// Map values
SIR.Position := PositionName;
SIR.Code := Code;
SIR.TU_ID := TU_ID;
SIR.Counter1 := Counter1;
SIR.Counter2 := Counter2;
SIR.Counter3 := Counter3;
SIR.Counter4 := Counter4;
SIR.Counter5 := Counter5;
SIR.eReturnCode := eReturnCode;

// Forward to ITC
F_ITC_SendSIR := fbITC_Manager.M_SendData(
					meChannel	:= eChannelSrc,
					mMsgType	:= E_ITC_MsgTypeConv.SCANNER_INFORMATION_REPORT,
					mpData		:= ADR(SIR),
					mLen		:= SIZEOF(SIR));

END_FUNCTION

// ---- 20_Product/10_BCF/11_Conv/11_Com/11_ITC/F_ITC_SendSNR.TcPOU
FUNCTION F_ITC_SendSNR : BOOL
(**************************************************************************************
 * 	Application		:	BoxControl Framework
 *	Revision		:	$Revision: 404529 $
 *	Revision date	:	$Date: 2018-04-23 08:21:38 +0200 (Mo., 23 Apr 2018) $
 *	Last changed by	:	$Author: b7bolm $
 *	URL				:	$URL: http://almscdc.swisslog.com/repo/SWPD/Development/BoxControlFramework/20_Release/trunk/01_Software/BCF/BCF/JumpStart/20_Product/10_App/11_Com/10_Lib/10_Conv/11_ITC/F_ITC_SendSNR.TcPOU $
 *
 *	Purpose			:	Wrap message - SNR
 *
 * ------------------------------------------------------------------------------------
 *	Copyright Swisslog [IP AG], Switzerland. All rights reserved.
 * 
 * ------------------------------------------------------------------------------------
 *	
 * 	Revision History: 
 *
 * 	VERSION			DATE			INITIALS			DESCRIPTION
 *	0.1				01.01.2001		swl					Example
 *
 **************************************************************************************)
VAR_INPUT
	eChannelSrc		: E_MFCS_Channel; // Source communicaton channel	
	PositionName	: STRING(Conveyor.POSITION_STRINGLENGTH); // Position
	TU_ID			: STRING(Conveyor.TU_ID_STRINGLENGTH); // TU ID
	eInfoCode		: E_ErrorConv; // Info Code
END_VAR
VAR
	SNR				: ST_ITC_SNR; 
END_VAR

// Map values
SNR.Position := PositionName;
SNR.TU_ID := TU_ID;
SNR.InfoCode := eInfoCode;

// Forward to ITC
F_ITC_SendSNR := fbITC_Manager.M_SendData(
					meChannel	:= eChannelSrc,
					mMsgType	:= E_ITC_MsgTypeConv.SCANNER_NO_READ_REPORT,
					mpData		:= ADR(SNR),
					mLen		:= SIZEOF(SNR));

END_FUNCTION

// ---- 20_Product/10_BCF/11_Conv/11_Com/11_ITC/F_ITC_SendTDR.TcPOU
FUNCTION F_ITC_SendTDR : BOOL
(**************************************************************************************
 * 	Application		:	BoxControl Framework
 *	Revision		:	$Revision: 404529 $
 *	Revision date	:	$Date: 2018-04-23 08:21:38 +0200 (Mo., 23 Apr 2018) $
 *	Last changed by	:	$Author: b7bolm $
 *	URL				:	$URL: http://almscdc.swisslog.com/repo/SWPD/Development/BoxControlFramework/20_Release/trunk/01_Software/BCF/BCF/JumpStart/20_Product/10_App/11_Com/10_Lib/10_Conv/11_ITC/F_ITC_SendTDR.TcPOU $
 *
 *	Purpose			:	Wrap message - TDR
 *
 * ------------------------------------------------------------------------------------
 *	Copyright Swisslog [IP AG], Switzerland. All rights reserved.
 * 
 * ------------------------------------------------------------------------------------
 *	
 * 	Revision History: 
 *
 * 	VERSION			DATE			INITIALS			DESCRIPTION
 *	0.1				01.01.2001		swl					Example
 *
 **************************************************************************************)
VAR_INPUT
	eChannelSrc		: E_MFCS_Channel; // Source communicaton channel	
	PositionName	: STRING(Conveyor.POSITION_STRINGLENGTH); // SIS MM-GGG-EEEE-FF-Z
	TU_ID			: STRING(Conveyor.TU_ID_STRINGLENGTH); // 18 Digit SSID
	AssignmentID	: UDINT; // assignment id
	MsgSequence		: INT; // MSG Sequence
	eReturnCode		: E_ErrorConv; // Return code
END_VAR
VAR
	TDR				: ST_ITC_TDR; 
END_VAR

// Map values
TDR.Position := PositionName;
TDR.TU_ID := TU_ID;
TDR.AssignmentID := AssignmentID;
TDR.MsgSequence := MsgSequence;
TDR.ReturnCode := eReturnCode;

// Forward to ITC
F_ITC_SendTDR := fbITC_Manager.M_SendData(
					meChannel	:= eChannelSrc,
					mMsgType	:= E_ITC_MsgTypeConv.TASK_DELETE_REPORT,
					mpData		:= ADR(TDR),
					mLen		:= SIZEOF(TDR));

END_FUNCTION

// ---- 20_Product/10_BCF/11_Conv/11_Com/11_ITC/F_ITC_SendTTC.TcPOU
FUNCTION F_ITC_SendTTC : BOOL
(**************************************************************************************
 * 	Application		:	BoxControl Framework
 *	Revision		:	$Revision: 404529 $
 *	Revision date	:	$Date: 2018-04-23 08:21:38 +0200 (Mo., 23 Apr 2018) $
 *	Last changed by	:	$Author: b7bolm $
 *	URL				:	$URL: http://almscdc.swisslog.com/repo/SWPD/Development/BoxControlFramework/20_Release/trunk/01_Software/BCF/BCF/JumpStart/20_Product/10_App/11_Com/10_Lib/10_Conv/11_ITC/F_ITC_SendTTC.TcPOU $
 *
 *	Purpose			:	Wrap message - TTC
 *
 * ------------------------------------------------------------------------------------
 *	Copyright Swisslog [IP AG], Switzerland. All rights reserved.
 * 
 * ------------------------------------------------------------------------------------
 *	
 * 	Revision History: 
 *
 * 	VERSION			DATE			INITIALS			DESCRIPTION
 *	0.1				01.01.2001		swl					Example
 *
 **************************************************************************************)
VAR_INPUT
	eChannelSrc		: E_MFCS_Channel; // Source communicaton channel		
	PositionName	: STRING(Conveyor.POSITION_STRINGLENGTH); // Position
	TU_DataIndex	: DINT; // TU-DataIndex
	MsgSequence		: INT; // Assignment message sequence
	TU_ID			: STRING(Conveyor.TU_ID_STRINGLENGTH); // 18 Digit SSID
	AssignmentID	: UDINT; // assignment id
	eReturnCode		: E_ErrorConv; // Return code
END_VAR
VAR
	TTC				: ST_ITC_TTC; 
END_VAR

// Map values
TTC.Position := PositionName;
TTC.TU_DataIndex := TU_DataIndex;
TTC.MsgSequence := MsgSequence;
TTC.TU_ID := TU_ID;
TTC.AssignmentID := AssignmentID;
TTC.ReturnCode := eReturnCode;

// Forward to ITC
F_ITC_SendTTC := fbITC_Manager.M_SendData(
					meChannel	:= eChannelSrc,
					mMsgType	:= E_ITC_MsgTypeConv.TRANSPORT_TASK_COMPLETE,
					mpData		:= ADR(TTC),
					mLen		:= SIZEOF(TTC));

END_FUNCTION

// ---- 20_Product/10_BCF/11_Conv/11_Com/11_ITC/F_ITC_SendTTQ.TcPOU
FUNCTION F_ITC_SendTTQ : BOOL
(**************************************************************************************
 * 	Application		:	BoxControl Framework
 *	Revision		:	$Revision: 404529 $
 *	Revision date	:	$Date: 2018-04-23 08:21:38 +0200 (Mo., 23 Apr 2018) $
 *	Last changed by	:	$Author: b7bolm $
 *	URL				:	$URL: http://almscdc.swisslog.com/repo/SWPD/Development/BoxControlFramework/20_Release/trunk/01_Software/BCF/BCF/JumpStart/20_Product/10_App/11_Com/10_Lib/10_Conv/11_ITC/F_ITC_SendTTQ.TcPOU $
 *
 *	Purpose			:	Wrap message - TTQ
 *
 * ------------------------------------------------------------------------------------
 *	Copyright Swisslog [IP AG], Switzerland. All rights reserved.
 * 
 * ------------------------------------------------------------------------------------
 *	
 * 	Revision History: 
 *
 * 	VERSION			DATE			INITIALS			DESCRIPTION
 *	0.1				01.01.2001		swl					Example
 *
 **************************************************************************************)
VAR_INPUT
	eChannelSrc		: E_MFCS_Channel; // Source communicaton channel	
	PositionName	: STRING(Conveyor.POSITION_STRINGLENGTH); // Position
	TU_DataIndex	: DINT; // TU-DataIndex
	TU_ID			: STRING(Conveyor.TU_ID_STRINGLENGTH); // TU ID
	NbrOfTT			: INT; // Number of TT's
	Label			: STRING(Conveyor.LABEL_LENGTH); // Label length
END_VAR
VAR
	TTQ				: ST_ITC_TTQ; 
END_VAR

// Map values
TTQ.Position := PositionName;
TTQ.TU_DataIndex := TU_DataIndex;
TTQ.TU_ID := TU_ID;
TTQ.NbrOfTT := NbrOfTT;
TTQ.Label := Label;

// Forward to ITC
F_ITC_SendTTQ := fbITC_Manager.M_SendData(
					meChannel	:= eChannelSrc,
					mMsgType	:= E_ITC_MsgTypeConv.TRANSPORT_TASK_REQUEST,
					mpData		:= ADR(TTQ),
					mLen		:= SIZEOF(TTQ));

END_FUNCTION

// ---- 20_Product/10_BCF/11_Conv/11_Com/11_ITC/F_ITC_SendTUR.TcPOU
FUNCTION F_ITC_SendTUR : BOOL
(**************************************************************************************
 * 	Application		:	BoxControl Framework
 *	Revision		:	$Revision: 416339 $
 *	Revision date	:	$Date: 2018-10-31 13:50:31 +0100 (Wed, 31 Oct 2018) $
 *	Last changed by	:	$Author: b7bolm $
 *	URL				:	$URL: http://almscdc.swisslog.com/repo/SWPD/Development/BoxControlFramework/20_Release/branches/R1.5.x/01_Software/BCF/BCF/JumpStart/20_Product/10_App/11_Com/10_Lib/10_Conv/11_ITC/F_ITC_SendTUR.TcPOU $
 *
 *	Purpose			:	Wrap message - TUR
 *
 * ------------------------------------------------------------------------------------
 *	Copyright Swisslog [IP AG], Switzerland. All rights reserved.
 * 
 * ------------------------------------------------------------------------------------
 *	
 * 	Revision History: 
 *
 * 	VERSION			DATE			INITIALS			DESCRIPTION
 *	0.1				01.01.2001		swl					Example
 *
 **************************************************************************************)
VAR_INPUT
	eChannelSrc				: E_MFCS_Channel; // Source communicaton channel	
	LastPositionName		: STRING(Conveyor.POSITION_STRINGLENGTH); // Position
	TU_DataIndex			: DINT; // Data index
	TU_ID					: STRING(Conveyor.TU_ID_STRINGLENGTH); // TU ID
	TU_Type					: INT; // TU Type
	AssignmentID			: UDINT; // Assignment ID
	Length					: INT; // Length
	Width					: INT; // Width
	Height					: INT; // Height
	Weight					: DINT; // Weight
	Orientation				: STRING(Conveyor.ORIENTATION_STRINGLENGTH); // 3 Digit orientation
	TU_Parameter			: INT; // TU Parameter
	IO_Data					: INT; // IO Data
	LowerLimit				: DINT; // Lower Limit
	UpperLimit				: DINT; // Upper Limit
	Sequence				: ULINT; // Global sequence identifier
	SubSequence				: DINT; // Position in the sequence
	SequenceSize			: DINT; // Number of TU's in the sequence
	GroupID					: ULINT; // Global group identifier 
	GroupSize				: DINT; // Number of TU's in the group ID
	DestinationSlot         : INT; // Logical sub destination of destination
	eReturnCode				: E_ErrorConv; // Return code
	NumberOfDestinations	: INT; // Number of Destinations
	Destination				: ARRAY [1..Conveyor.NUMBER_OF_DESTINATIONS] OF STRING(Conveyor.POSITION_STRINGLENGTH); // Array of SIS Destinations
END_VAR
VAR
	TUR						: ST_ITC_TUR; 
END_VAR

// Map values
TUR.Position := LastPositionName;
TUR.TU_DataIndex := TU_DataIndex;
TUR.TU_ID := TU_ID;
TUR.TU_Type := TU_Type;
TUR.AssignmentID := AssignmentID;
TUR.Length := Length;
TUR.Width := Width;
TUR.Height := Height;
TUR.Weight := Weight;
TUR.Orientation := Orientation;
TUR.TU_Parameter := TU_Parameter;
TUR.IO_Data := IO_Data;
TUR.LowerLimit := LowerLimit;
TUR.UpperLimit := UpperLimit;
TUR.Sequence := Sequence;
TUR.SubSequence := SubSequence;
TUR.SequenceSize := SequenceSize;
TUR.GroupID := GroupID;
TUR.GroupSize := GroupSize;
TUR.DestinationSlot := DestinationSlot;
TUR.ReturnCode := eReturnCode;
TUR.NumberOfDestinations := NumberOfDestinations;
TUR.Destination := Destination;

// Forward to ITC
F_ITC_SendTUR := fbITC_Manager.M_SendData(
					meChannel	:= eChannelSrc,
					mMsgType	:= E_ITC_MsgTypeConv.TRANSPORT_UNIT_REPORT,
					mpData		:= ADR(TUR),
					mLen		:= SIZEOF(TUR));

END_FUNCTION

// ---- 20_Product/10_BCF/11_Conv/11_Com/13_Sub-Sub/FB_STI_SendReceiveTU_Data_6_0.TcPOU
FUNCTION_BLOCK FB_STI_SendReceiveTU_Data_6_0
(**************************************************************************************
 * 	Application		:	BoxControl Framework
 *	Revision		:	$Revision: 404529 $
 *	Revision date	:	$Date: 2018-04-23 08:21:38 +0200 (Mo., 23 Apr 2018) $
 *	Last changed by	:	$Author: b7bolm $
 *	URL				:	$URL: http://almscdc.swisslog.com/repo/SWPD/Development/BoxControlFramework/20_Release/trunk/01_Software/BCF/BCF/JumpStart/20_Product/10_App/11_Com/10_Lib/10_Conv/13_Sub-Sub/FB_STI_SendReceiveTU_Data_6_0.TcPOU $
 *
 *	Purpose			:	Sends and Receive TU-data to/from other SubSystem via TTA
 *
 * ------------------------------------------------------------------------------------
 *	Copyright Swisslog [IP AG], Switzerland. All rights reserved.
 * 
 * ------------------------------------------------------------------------------------
 *	
 * 	Revision History: 
 *
 * 	VERSION			DATE			INITIALS			DESCRIPTION
 *	0.1				01.01.2001		swl					Example
 *
 **************************************************************************************)
VAR_INPUT
	PositionSubSystem		: STRING(SIS_6_0.POSITION_STRINGLENGTH); // SIS-Position of SubSystem
	ConfigSIS_MsgManager	: ST_CFG_SIS_MsgManager_6_0; // Configuration
END_VAR
VAR
	Init					: BOOL := FALSE; // Instance is initialized
	fbMFCS_SIS_Sub			: FB_SIS_MsgManager_6_0; // Instance of SIS-driver
	TTA						: ST_TTA_6_0; // TTA structure
	SendTelegram			: ARRAY [1..MAX_STREAM_LENGTH] OF BYTE; // Send telegram
END_VAR
VAR CONSTANT
	MAX_STREAM_LENGTH		: UDINT := 30000; // Number of bytes of one message
END_VAR

(**************************************************************************************************************
   Initialization
***************************************************************************************************************)
A_Init();


(**************************************************************************************************************
   Call SIS-driver
***************************************************************************************************************)
fbMFCS_SIS_Sub.M_CallCommunicationService();

ACTION A_Init:
(**************************************************************************************
 * 	NAME		A_Init
 * 	FUNCTION	Initialize FB
 **************************************************************************************)
// If instance is not initialized or init is forced
IF NOT Init THEN
	
	// Activate configuration
	fbMFCS_SIS_Sub.Config := ConfigSIS_MsgManager;
	
	// Init done
    Init := TRUE;
END_IF
END_ACTION

METHOD M_SendTTA : BOOL
(**************************************************************************************
 * 	Application		:	BoxControl Framework
 *	Revision		:	$Revision: 404529 $
 *	Revision date	:	$Date: 2018-04-23 08:21:38 +0200 (Mo., 23 Apr 2018) $
 *	Last changed by	:	$Author: b7bolm $
 *	URL				:	$URL: http://almscdc.swisslog.com/repo/SWPD/Development/BoxControlFramework/20_Release/trunk/01_Software/BCF/BCF/JumpStart/20_Product/10_App/11_Com/10_Lib/10_Conv/13_Sub-Sub/FB_STI_SendReceiveTU_Data_6_0.TcPOU $
 *
 *	Purpose			:	Send TTA
 *
 * ------------------------------------------------------------------------------------
 *	Copyright Swisslog [IP AG], Switzerland. All rights reserved.
 * 
 * ------------------------------------------------------------------------------------
 *	
 * 	Revision History: 
 *
 * 	VERSION			DATE			INITIALS			DESCRIPTION
 *	0.1				01.01.2001		swl					Example
 *
 **************************************************************************************)
VAR_INPUT
 	mTU_DataIndex		: DINT;
END_VAR
VAR
	mIdx				: INT;
	mWritePointer		: UDINT;
END_VAR
(**************************************************************************************************************
 	Formatting data
***************************************************************************************************************)
TTA.Position := F_StuffString(
					InputString 	:= PositionSubSystem, 
					StringLength	:= SIS_6_0.POSITION_STRINGLENGTH, 
					StuffCharacter 	:= '0',
					LeftAligned		:= FALSE);
					
TTA.TU_DataIndex := F_StuffString(
					InputString 	:= '0', 
					StringLength	:= SIS_6_0.TU_DATAINDEX_STRINGLENGTH, 
					StuffCharacter 	:= '0',
					LeftAligned		:= FALSE);
					
TTA.MsgSequence := F_StuffString(
					InputString 	:= '0', 
					StringLength	:= SIS_6_0.MSG_SEQUENCE_STRINGLENGTH, 
					StuffCharacter 	:= '0',
					LeftAligned		:= FALSE);

TTA.TU_ID := F_StuffString(
					InputString 	:= TU_DataTable[mTU_DataIndex].TU_ID.ASCII, 
					StringLength	:= SIS_6_0.TU_ID_STRINGLENGTH, 
					StuffCharacter 	:= ' ',
					LeftAligned		:= FALSE);
					
TTA.TU_Type := F_StuffString(
					InputString 	:= INT_TO_STRING(TU_DataTable[mTU_DataIndex].DataSet.TU_Type), 
					StringLength	:= SIS_6_0.TU_TYPE_STRINGLENGTH, 
					StuffCharacter 	:= '0',
					LeftAligned		:= FALSE);
					
TTA.AssignmentID := F_StuffString(
					InputString 	:= UDINT_TO_STRING(TU_DataTable[mTU_DataIndex].AssignmentID), 
					StringLength	:= SIS_6_0.ASSIGNMENT_ID_STRINGLENGTH, 
					StuffCharacter 	:= '0',
					LeftAligned		:= FALSE);
					
TTA.Length := F_StuffString(
					InputString 	:= INT_TO_STRING(TU_DataTable[mTU_DataIndex].DataSet.Dimension.Length), 
					StringLength	:= SIS_6_0.DIMENSIONS, 
					StuffCharacter 	:= '0',
					LeftAligned		:= FALSE);
					
TTA.Width := F_StuffString(
					InputString 	:= INT_TO_STRING(TU_DataTable[mTU_DataIndex].DataSet.Dimension.Width), 
					StringLength	:= SIS_6_0.DIMENSIONS, 
					StuffCharacter 	:= '0',
					LeftAligned		:= FALSE);
					
TTA.Height := F_StuffString(
					InputString 	:= INT_TO_STRING(TU_DataTable[mTU_DataIndex].DataSet.Dimension.Height), 
					StringLength	:= SIS_6_0.DIMENSIONS, 
					StuffCharacter 	:= '0',
					LeftAligned		:= FALSE);
					
TTA.Weight := F_StuffString(
					InputString 	:= DINT_TO_STRING(TU_DataTable[mTU_DataIndex].DataSet.Dimension.Weight), 
					StringLength	:= SIS_6_0.TTA_WEIGHT, 
					StuffCharacter 	:= '0',
					LeftAligned		:= FALSE);
					
TTA.Orientation := F_StuffString(
					InputString 	:= TU_DataTable[mTU_DataIndex].DataSet.Orientation, 
					StringLength	:= SIS_6_0.TTA_ORIENTATION, 
					StuffCharacter 	:= '0',
					LeftAligned		:= FALSE);

TTA.TU_Parameter := F_StuffString(
					InputString 	:= INT_TO_STRING(TU_DataTable[mTU_DataIndex].DataSet.TU_Parameter), 
					StringLength	:= SIS_6_0.TTA_TU_PARAMETER, 
					StuffCharacter 	:= '0',
					LeftAligned		:= FALSE);
					
TTA.IO_Data := F_StuffString(
					InputString 	:= INT_TO_STRING(TU_DataTable[mTU_DataIndex].DataSet.IO_Data), 
					StringLength	:= SIS_6_0.TTA_IO_DATA_STRINGLENGTH, 
					StuffCharacter 	:= '0',
					LeftAligned		:= FALSE);
					
TTA.LowerLimit := F_StuffString(
					InputString 	:= DINT_TO_STRING(TU_DataTable[mTU_DataIndex].DataSet.LowerLimit), 
					StringLength	:= SIS_6_0.TTA_LOWER_LIMIT_STRINGLENGTH, 
					StuffCharacter 	:= '0',
					LeftAligned		:= FALSE);
					
TTA.UpperLimit := F_StuffString(
					InputString 	:= DINT_TO_STRING(TU_DataTable[mTU_DataIndex].DataSet.UpperLimit), 
					StringLength	:= SIS_6_0.TTA_UPPER_LIMIT_STRINGLENGTH, 
					StuffCharacter 	:= '0',
					LeftAligned		:= FALSE);
					
TTA.GroupInfo := F_StuffString(
					InputString 	:= ULINT_TO_STRING(TU_DataTable[mTU_DataIndex].DataSet.GroupID), 
					StringLength	:= SIS_6_0.TTA_GROUPINFO_STRINGLENGTH, 
					StuffCharacter 	:= '0',
					LeftAligned		:= FALSE);
					
TTA.Sequence := F_StuffString(
					InputString 	:= ULINT_TO_STRING(TU_DataTable[mTU_DataIndex].DataSet.Sequence), 
					StringLength	:= SIS_6_0.TTA_SEQUENCE_STRINGLENGTH, 
					StuffCharacter 	:= '0',
					LeftAligned		:= FALSE);
					
TTA.NumberInSequence := F_StuffString(
					InputString 	:= DINT_TO_STRING(TU_DataTable[mTU_DataIndex].DataSet.SubSequence), 
					StringLength	:= SIS_6_0.TTA_NO_IN_SEQUENCE_STRINGLENGTH, 
					StuffCharacter 	:= '0',
					LeftAligned		:= FALSE);
					
TTA.NumberOfDestinations := F_StuffString(
					InputString 	:= INT_TO_STRING(TU_DataTable[mTU_DataIndex].DataSet.NumberOfDest), 
					StringLength	:= SIS_6_0.TTA_NO_OF_DESTINATIONS_STRINGLENGTH, 
					StuffCharacter 	:= '0',
					LeftAligned		:= FALSE);
					
FOR mIdx := 1 TO TU_DataTable[mTU_DataIndex].DataSet.NumberOfDest DO
	TTA.Destination[mIdx] := F_StuffString(
					InputString 	:= TU_DataTable[mTU_DataIndex].Destination[mIdx].PositionName, 
					StringLength	:= SIS_6_0.POSITION_STRINGLENGTH, 
					StuffCharacter 	:= '0',
					LeftAligned		:= FALSE);
END_FOR
					
					
(**************************************************************************************************************
 	Build string and add to Base Driver
***************************************************************************************************************)
MEMSET(destAddr := ADR(SendTelegram), 0, SIZEOF(SendTelegram));
mWritePointer := 0;

F_AssembleByteStream(
	pSrc 			:= ADR('TTA'), 
	SrcLen 			:= 3, 
	pDest 			:= ADR(SendTelegram), 
	DestLen 		:= SIZEOF(SendTelegram), 
	WritePointer	:= mWritePointer);
	
F_AssembleByteStream(
	pSrc 			:= ADR(TTA.Position), 
	SrcLen 			:= INT_TO_UDINT(LEN(TTA.Position)), 
	pDest 			:= ADR(SendTelegram), 
	DestLen 		:= SIZEOF(SendTelegram), 
	WritePointer	:= mWritePointer);
	
F_AssembleByteStream(
	pSrc 			:= ADR(TTA.TU_DataIndex), 
	SrcLen 			:= INT_TO_UDINT(LEN(TTA.TU_DataIndex)), 
	pDest 			:= ADR(SendTelegram), 
	DestLen 		:= SIZEOF(SendTelegram), 
	WritePointer	:= mWritePointer);
	
F_AssembleByteStream(
	pSrc 			:= ADR(TTA.MsgSequence), 
	SrcLen 			:= INT_TO_UDINT(LEN(TTA.MsgSequence)), 
	pDest 			:= ADR(SendTelegram), 
	DestLen 		:= SIZEOF(SendTelegram), 
	WritePointer	:= mWritePointer);
	
F_AssembleByteStream(
	pSrc 			:= ADR(TTA.TU_ID), 
	SrcLen 			:= INT_TO_UDINT(LEN(TTA.TU_ID)), 
	pDest 			:= ADR(SendTelegram), 
	DestLen 		:= SIZEOF(SendTelegram), 
	WritePointer	:= mWritePointer);
	
F_AssembleByteStream(
	pSrc 			:= ADR(TTA.TU_Type), 
	SrcLen 			:= INT_TO_UDINT(LEN(TTA.TU_Type)), 
	pDest 			:= ADR(SendTelegram), 
	DestLen 		:= SIZEOF(SendTelegram), 
	WritePointer	:= mWritePointer);	
	
F_AssembleByteStream(
	pSrc 			:= ADR(TTA.AssignmentID), 
	SrcLen 			:= INT_TO_UDINT(LEN(TTA.AssignmentID)), 
	pDest 			:= ADR(SendTelegram), 
	DestLen 		:= SIZEOF(SendTelegram), 
	WritePointer	:= mWritePointer);		
	
F_AssembleByteStream(
	pSrc 			:= ADR(TTA.Length), 
	SrcLen 			:= INT_TO_UDINT(LEN(TTA.Length)), 
	pDest 			:= ADR(SendTelegram), 
	DestLen 		:= SIZEOF(SendTelegram), 
	WritePointer	:= mWritePointer);

F_AssembleByteStream(
	pSrc 			:= ADR(TTA.Width), 
	SrcLen 			:= INT_TO_UDINT(LEN(TTA.Width)), 
	pDest 			:= ADR(SendTelegram), 
	DestLen 		:= SIZEOF(SendTelegram), 
	WritePointer	:= mWritePointer);
	
F_AssembleByteStream(
	pSrc 			:= ADR(TTA.Height), 
	SrcLen 			:= INT_TO_UDINT(LEN(TTA.Height)), 
	pDest 			:= ADR(SendTelegram), 
	DestLen 		:= SIZEOF(SendTelegram), 
	WritePointer	:= mWritePointer);
	
F_AssembleByteStream(
	pSrc 			:= ADR(TTA.Weight), 
	SrcLen 			:= INT_TO_UDINT(LEN(TTA.Weight)), 
	pDest 			:= ADR(SendTelegram), 
	DestLen 		:= SIZEOF(SendTelegram), 
	WritePointer	:= mWritePointer);
		
F_AssembleByteStream(
	pSrc 			:= ADR(TTA.Orientation), 
	SrcLen 			:= INT_TO_UDINT(LEN(TTA.Orientation)), 
	pDest 			:= ADR(SendTelegram), 
	DestLen 		:= SIZEOF(SendTelegram), 
	WritePointer	:= mWritePointer);
	
F_AssembleByteStream(
	pSrc 			:= ADR(TTA.TU_Parameter), 
	SrcLen 			:= INT_TO_UDINT(LEN(TTA.TU_Parameter)), 
	pDest 			:= ADR(SendTelegram), 
	DestLen 		:= SIZEOF(SendTelegram), 
	WritePointer	:= mWritePointer);	
	
F_AssembleByteStream(
	pSrc 			:= ADR(TTA.IO_Data), 
	SrcLen 			:= INT_TO_UDINT(LEN(TTA.IO_Data)), 
	pDest 			:= ADR(SendTelegram), 
	DestLen 		:= SIZEOF(SendTelegram), 
	WritePointer	:= mWritePointer);
	
F_AssembleByteStream(
	pSrc 			:= ADR(TTA.LowerLimit), 
	SrcLen 			:= INT_TO_UDINT(LEN(TTA.LowerLimit)), 
	pDest 			:= ADR(SendTelegram), 
	DestLen 		:= SIZEOF(SendTelegram), 
	WritePointer	:= mWritePointer);
	
F_AssembleByteStream(
	pSrc 			:= ADR(TTA.UpperLimit), 
	SrcLen 			:= INT_TO_UDINT(LEN(TTA.UpperLimit)), 
	pDest 			:= ADR(SendTelegram), 
	DestLen 		:= SIZEOF(SendTelegram), 
	WritePointer	:= mWritePointer);
	
F_AssembleByteStream(
	pSrc 			:= ADR(TTA.GroupInfo), 
	SrcLen 			:= INT_TO_UDINT(LEN(TTA.GroupInfo)), 
	pDest 			:= ADR(SendTelegram), 
	DestLen 		:= SIZEOF(SendTelegram), 
	WritePointer	:= mWritePointer);
	
F_AssembleByteStream(
	pSrc 			:= ADR(TTA.Sequence), 
	SrcLen 			:= INT_TO_UDINT(LEN(TTA.Sequence)), 
	pDest 			:= ADR(SendTelegram), 
	DestLen 		:= SIZEOF(SendTelegram), 
	WritePointer	:= mWritePointer);
	
F_AssembleByteStream(
	pSrc 			:= ADR(TTA.NumberInSequence), 
	SrcLen 			:= INT_TO_UDINT(LEN(TTA.NumberInSequence)), 
	pDest 			:= ADR(SendTelegram), 
	DestLen 		:= SIZEOF(SendTelegram), 
	WritePointer	:= mWritePointer);	

F_AssembleByteStream(
	pSrc 			:= ADR(TTA.NumberOfDestinations), 
	SrcLen 			:= INT_TO_UDINT(LEN(TTA.NumberOfDestinations)), 
	pDest 			:= ADR(SendTelegram), 
	DestLen 		:= SIZEOF(SendTelegram), 
	WritePointer	:= mWritePointer);	

FOR mIdx := 1 TO TU_DataTable[mTU_DataIndex].DataSet.NumberOfDest DO
	F_AssembleByteStream(
		pSrc 			:= ADR(TTA.Destination[mIdx]), 
		SrcLen 			:= INT_TO_UDINT(LEN(TTA.Destination[mIdx])), 
		pDest 			:= ADR(SendTelegram), 
		DestLen 		:= SIZEOF(SendTelegram), 
		WritePointer	:= mWritePointer);	
END_FOR	

M_SendTTA := fbMFCS_SIS_Sub.M_SendAppData(pData := ADR(SendTelegram), DataLen := mWritePointer);
END_METHOD

END_FUNCTION_BLOCK

// ---- 20_Product/10_BCF/11_Conv/11_Com/13_Sub-Sub/FB_STI_SendReceiveTU_Data_6_1.TcPOU
FUNCTION_BLOCK FB_STI_SendReceiveTU_Data_6_1
(**************************************************************************************
 * 	Application		:	BoxControl Framework
 *	Revision		:	$Revision: 404529 $
 *	Revision date	:	$Date: 2018-04-23 08:21:38 +0200 (Mo., 23 Apr 2018) $
 *	Last changed by	:	$Author: b7bolm $
 *	URL				:	$URL: http://almscdc.swisslog.com/repo/SWPD/Development/BoxControlFramework/20_Release/trunk/01_Software/BCF/BCF/JumpStart/20_Product/10_App/11_Com/10_Lib/10_Conv/13_Sub-Sub/FB_STI_SendReceiveTU_Data_6_1.TcPOU $
 *
 *	Purpose			:	Sends and Receive TU-data to/from other SubSystem via TTA
 *
 * ------------------------------------------------------------------------------------
 *	Copyright Swisslog [IP AG], Switzerland. All rights reserved.
 * 
 * ------------------------------------------------------------------------------------
 *	
 * 	Revision History: 
 *
 * 	VERSION			DATE			INITIALS			DESCRIPTION
 *	0.1				01.01.2001		swl					Example
 *
 **************************************************************************************)
VAR_INPUT
	PositionSubSystem		: STRING(SIS_6_1.POSITION_STRINGLENGTH); // SIS-Position of SubSystem
	ConfigSIS_MsgManager	: ST_CFG_SIS_MsgManager_6_1; // Configuration
END_VAR
VAR
	Init					: BOOL := FALSE; // Instance is initialized
	fbMFCS_SIS_Sub			: FB_SIS_MsgManager_6_1; // Instance of SIS-driver
	TTA						: ST_TTA_6_1; // TTA structure
	SendTelegram			: ARRAY [1..MAX_STREAM_LENGTH] OF BYTE; // Send telegram
END_VAR
VAR CONSTANT
	MAX_STREAM_LENGTH		: UDINT := 30000; // Number of bytes of one message
END_VAR

(**************************************************************************************************************
   Initialization
***************************************************************************************************************)
A_Init();


(**************************************************************************************************************
   Call SIS-driver
***************************************************************************************************************)
fbMFCS_SIS_Sub.M_CallCommunicationService();

ACTION A_Init:
(**************************************************************************************
 * 	NAME		A_Init
 * 	FUNCTION	Initialize FB
 **************************************************************************************)
// If instance is not initialized or init is forced
IF NOT Init THEN
	
	// Activate configuration
	fbMFCS_SIS_Sub.Config := ConfigSIS_MsgManager;
	
	// Init done
    Init := TRUE;
END_IF
END_ACTION

METHOD M_SendTTA : BOOL
(**************************************************************************************
 * 	Application		:	BoxControl Framework
 *	Revision		:	$Revision: 404529 $
 *	Revision date	:	$Date: 2018-04-23 08:21:38 +0200 (Mo., 23 Apr 2018) $
 *	Last changed by	:	$Author: b7bolm $
 *	URL				:	$URL: http://almscdc.swisslog.com/repo/SWPD/Development/BoxControlFramework/20_Release/trunk/01_Software/BCF/BCF/JumpStart/20_Product/10_App/11_Com/10_Lib/10_Conv/13_Sub-Sub/FB_STI_SendReceiveTU_Data_6_1.TcPOU $
 *
 *	Purpose			:	Send TTA
 *
 * ------------------------------------------------------------------------------------
 *	Copyright Swisslog [IP AG], Switzerland. All rights reserved.
 * 
 * ------------------------------------------------------------------------------------
 *	
 * 	Revision History: 
 *
 * 	VERSION			DATE			INITIALS			DESCRIPTION
 *	0.1				01.01.2001		swl					Example
 *
 **************************************************************************************)
VAR_INPUT
 	mTU_DataIndex		: DINT;
END_VAR
VAR
	mIdx				: INT;
	mWritePointer		: UDINT;
END_VAR
(**************************************************************************************************************
 	Formatting data
***************************************************************************************************************)
TTA.Position := F_StuffString(
					InputString 	:= PositionSubSystem, 
					StringLength	:= SIS_6_1.POSITION_STRINGLENGTH, 
					StuffCharacter 	:= '0',
					LeftAligned		:= FALSE);
					
TTA.TU_DataIndex := F_StuffString(
						InputString 	:= '0', 
						StringLength	:= SIS_6_1.TU_DATAINDEX_STRINGLENGTH, 
						StuffCharacter 	:= '0',
						LeftAligned		:= FALSE);
					
TTA.MsgSequence := F_StuffString(
					InputString 	:= '0', 
					StringLength	:= SIS_6_1.MSG_SEQUENCE_STRINGLENGTH, 
					StuffCharacter 	:= '0',
					LeftAligned		:= FALSE);

TTA.TU_ID := F_StuffString(
				InputString 	:= TU_DataTable[mTU_DataIndex].TU_ID.ASCII, 
				StringLength	:= SIS_6_1.TU_ID_STRINGLENGTH, 
				StuffCharacter 	:= ' ',
				LeftAligned		:= FALSE);
					
TTA.TU_Type := F_StuffString(
				InputString 	:= INT_TO_STRING(TU_DataTable[mTU_DataIndex].DataSet.TU_Type), 
				StringLength	:= SIS_6_1.TU_TYPE_STRINGLENGTH, 
				StuffCharacter 	:= '0',
				LeftAligned		:= FALSE);
					
TTA.AssignmentID := F_StuffString(
						InputString 	:= UDINT_TO_STRING(TU_DataTable[mTU_DataIndex].AssignmentID), 
						StringLength	:= SIS_6_1.ASSIGNMENT_ID_STRINGLENGTH, 
						StuffCharacter 	:= '0',
						LeftAligned		:= FALSE);
					
TTA.Length := F_StuffString(
				InputString 	:= INT_TO_STRING(TU_DataTable[mTU_DataIndex].DataSet.Dimension.Length), 
				StringLength	:= SIS_6_1.DIMENSIONS, 
				StuffCharacter 	:= '0',
				LeftAligned		:= FALSE);
					
TTA.Width := F_StuffString(
				InputString 	:= INT_TO_STRING(TU_DataTable[mTU_DataIndex].DataSet.Dimension.Width), 
				StringLength	:= SIS_6_1.DIMENSIONS, 
				StuffCharacter 	:= '0',
				LeftAligned		:= FALSE);
					
TTA.Height := F_StuffString(
				InputString 	:= INT_TO_STRING(TU_DataTable[mTU_DataIndex].DataSet.Dimension.Height), 
				StringLength	:= SIS_6_1.DIMENSIONS, 
				StuffCharacter 	:= '0',
				LeftAligned		:= FALSE);
					
TTA.Weight := F_StuffString(
				InputString 	:= DINT_TO_STRING(TU_DataTable[mTU_DataIndex].DataSet.Dimension.Weight), 
				StringLength	:= SIS_6_1.TTA_WEIGHT, 
				StuffCharacter 	:= '0',
				LeftAligned		:= FALSE);
					
TTA.Orientation := F_StuffString(
					InputString 	:= TU_DataTable[mTU_DataIndex].DataSet.Orientation, 
					StringLength	:= SIS_6_1.TTA_ORIENTATION, 
					StuffCharacter 	:= '0',
					LeftAligned		:= FALSE);

TTA.TU_Parameter := F_StuffString(
						InputString 	:= INT_TO_STRING(TU_DataTable[mTU_DataIndex].DataSet.TU_Parameter), 
						StringLength	:= SIS_6_1.TTA_TU_PARAMETER, 
						StuffCharacter 	:= '0',
						LeftAligned		:= FALSE);
					
TTA.IO_Data := F_StuffString(
					InputString 	:= INT_TO_STRING(TU_DataTable[mTU_DataIndex].DataSet.IO_Data), 
					StringLength	:= SIS_6_1.TTA_IO_DATA_STRINGLENGTH, 
					StuffCharacter 	:= '0',
					LeftAligned		:= FALSE);
					
TTA.LowerLimit := F_StuffString(
					InputString 	:= DINT_TO_STRING(TU_DataTable[mTU_DataIndex].DataSet.LowerLimit), 
					StringLength	:= SIS_6_1.TTA_LOWER_LIMIT_STRINGLENGTH, 
					StuffCharacter 	:= '0',
					LeftAligned		:= FALSE);
					
TTA.UpperLimit := F_StuffString(
					InputString 	:= DINT_TO_STRING(TU_DataTable[mTU_DataIndex].DataSet.UpperLimit), 
					StringLength	:= SIS_6_1.TTA_UPPER_LIMIT_STRINGLENGTH, 
					StuffCharacter 	:= '0',
					LeftAligned		:= FALSE);
					
TTA.Sequence := F_StuffString(
					InputString 	:= ULINT_TO_STRING(TU_DataTable[mTU_DataIndex].DataSet.Sequence), 
					StringLength	:= SIS_6_1.SEQUENCE_STRINGLENGTH, 
					StuffCharacter 	:= '0',
					LeftAligned		:= FALSE);

TTA.SubSequence := F_StuffString(
						InputString 	:= DINT_TO_STRING(TU_DataTable[mTU_DataIndex].DataSet.SubSequence), 
						StringLength	:= SIS_6_1.SUBSEQUENCE_STRINGLENGTH, 
						StuffCharacter 	:= '0',
						LeftAligned		:= FALSE);

TTA.SequenceSize := F_StuffString(
						InputString 	:= DINT_TO_STRING(TU_DataTable[mTU_DataIndex].DataSet.SequenceSize), 
						StringLength	:= SIS_6_1.SEQUENCE_SIZE_STRINGLENGTH, 
						StuffCharacter 	:= '0',
						LeftAligned		:= FALSE);

TTA.GroupID := F_StuffString(
				InputString 	:= ULINT_TO_STRING(TU_DataTable[mTU_DataIndex].DataSet.GroupID), 
				StringLength	:= SIS_6_1.GROUP_ID_STRINGLENGTH, 
				StuffCharacter 	:= '0',
				LeftAligned		:= FALSE);

TTA.GroupSize := F_StuffString(
					InputString 	:= DINT_TO_STRING(TU_DataTable[mTU_DataIndex].DataSet.GroupSize), 
					StringLength	:= SIS_6_1.GROUP_SIZE_STRINGLENGTH, 
					StuffCharacter 	:= '0',
					LeftAligned		:= FALSE);

TTA.DestinationSlot := F_StuffString(
							InputString 	:= INT_TO_STRING(TU_DataTable[mTU_DataIndex].DataSet.DestinationSlot), 
							StringLength	:= SIS_6_1.DESTINATION_SLOT_STRINGLENGTH, 
							StuffCharacter 	:= '0',
							LeftAligned		:= FALSE);
					
TTA.NumberOfDestinations := F_StuffString(
								InputString 	:= INT_TO_STRING(TU_DataTable[mTU_DataIndex].DataSet.NumberOfDest), 
								StringLength	:= SIS_6_1.TTA_NO_OF_DESTINATIONS_STRINGLENGTH, 
								StuffCharacter 	:= '0',
								LeftAligned		:= FALSE);
					
FOR mIdx := 1 TO TU_DataTable[mTU_DataIndex].DataSet.NumberOfDest DO
	TTA.Destination[mIdx] := F_StuffString(
								InputString 	:= TU_DataTable[mTU_DataIndex].Destination[mIdx].PositionName, 
								StringLength	:= SIS_6_1.POSITION_STRINGLENGTH, 
								StuffCharacter 	:= '0',
								LeftAligned		:= FALSE);
END_FOR
					
					
(**************************************************************************************************************
 	Build string and add to Base Driver
***************************************************************************************************************)
MEMSET(destAddr := ADR(SendTelegram), 0, SIZEOF(SendTelegram));
mWritePointer := 0;

F_AssembleByteStream(
	pSrc 			:= ADR('TTA'), 
	SrcLen 			:= 3, 
	pDest 			:= ADR(SendTelegram), 
	DestLen 		:= SIZEOF(SendTelegram), 
	WritePointer	:= mWritePointer);
	
F_AssembleByteStream(
	pSrc 			:= ADR(TTA.Position), 
	SrcLen 			:= INT_TO_UDINT(LEN(TTA.Position)), 
	pDest 			:= ADR(SendTelegram), 
	DestLen 		:= SIZEOF(SendTelegram), 
	WritePointer	:= mWritePointer);
	
F_AssembleByteStream(
	pSrc 			:= ADR(TTA.TU_DataIndex), 
	SrcLen 			:= INT_TO_UDINT(LEN(TTA.TU_DataIndex)), 
	pDest 			:= ADR(SendTelegram), 
	DestLen 		:= SIZEOF(SendTelegram), 
	WritePointer	:= mWritePointer);
	
F_AssembleByteStream(
	pSrc 			:= ADR(TTA.MsgSequence), 
	SrcLen 			:= INT_TO_UDINT(LEN(TTA.MsgSequence)), 
	pDest 			:= ADR(SendTelegram), 
	DestLen 		:= SIZEOF(SendTelegram), 
	WritePointer	:= mWritePointer);
	
F_AssembleByteStream(
	pSrc 			:= ADR(TTA.TU_ID), 
	SrcLen 			:= INT_TO_UDINT(LEN(TTA.TU_ID)), 
	pDest 			:= ADR(SendTelegram), 
	DestLen 		:= SIZEOF(SendTelegram), 
	WritePointer	:= mWritePointer);
	
F_AssembleByteStream(
	pSrc 			:= ADR(TTA.TU_Type), 
	SrcLen 			:= INT_TO_UDINT(LEN(TTA.TU_Type)), 
	pDest 			:= ADR(SendTelegram), 
	DestLen 		:= SIZEOF(SendTelegram), 
	WritePointer	:= mWritePointer);	
	
F_AssembleByteStream(
	pSrc 			:= ADR(TTA.AssignmentID), 
	SrcLen 			:= INT_TO_UDINT(LEN(TTA.AssignmentID)), 
	pDest 			:= ADR(SendTelegram), 
	DestLen 		:= SIZEOF(SendTelegram), 
	WritePointer	:= mWritePointer);		
	
F_AssembleByteStream(
	pSrc 			:= ADR(TTA.Length), 
	SrcLen 			:= INT_TO_UDINT(LEN(TTA.Length)), 
	pDest 			:= ADR(SendTelegram), 
	DestLen 		:= SIZEOF(SendTelegram), 
	WritePointer	:= mWritePointer);

F_AssembleByteStream(
	pSrc 			:= ADR(TTA.Width), 
	SrcLen 			:= INT_TO_UDINT(LEN(TTA.Width)), 
	pDest 			:= ADR(SendTelegram), 
	DestLen 		:= SIZEOF(SendTelegram), 
	WritePointer	:= mWritePointer);
	
F_AssembleByteStream(
	pSrc 			:= ADR(TTA.Height), 
	SrcLen 			:= INT_TO_UDINT(LEN(TTA.Height)), 
	pDest 			:= ADR(SendTelegram), 
	DestLen 		:= SIZEOF(SendTelegram), 
	WritePointer	:= mWritePointer);
	
F_AssembleByteStream(
	pSrc 			:= ADR(TTA.Weight), 
	SrcLen 			:= INT_TO_UDINT(LEN(TTA.Weight)), 
	pDest 			:= ADR(SendTelegram), 
	DestLen 		:= SIZEOF(SendTelegram), 
	WritePointer	:= mWritePointer);
		
F_AssembleByteStream(
	pSrc 			:= ADR(TTA.Orientation), 
	SrcLen 			:= INT_TO_UDINT(LEN(TTA.Orientation)), 
	pDest 			:= ADR(SendTelegram), 
	DestLen 		:= SIZEOF(SendTelegram), 
	WritePointer	:= mWritePointer);
	
F_AssembleByteStream(
	pSrc 			:= ADR(TTA.TU_Parameter), 
	SrcLen 			:= INT_TO_UDINT(LEN(TTA.TU_Parameter)), 
	pDest 			:= ADR(SendTelegram), 
	DestLen 		:= SIZEOF(SendTelegram), 
	WritePointer	:= mWritePointer);	
	
F_AssembleByteStream(
	pSrc 			:= ADR(TTA.IO_Data), 
	SrcLen 			:= INT_TO_UDINT(LEN(TTA.IO_Data)), 
	pDest 			:= ADR(SendTelegram), 
	DestLen 		:= SIZEOF(SendTelegram), 
	WritePointer	:= mWritePointer);
	
F_AssembleByteStream(
	pSrc 			:= ADR(TTA.LowerLimit), 
	SrcLen 			:= INT_TO_UDINT(LEN(TTA.LowerLimit)), 
	pDest 			:= ADR(SendTelegram), 
	DestLen 		:= SIZEOF(SendTelegram), 
	WritePointer	:= mWritePointer);
	
F_AssembleByteStream(
	pSrc 			:= ADR(TTA.UpperLimit), 
	SrcLen 			:= INT_TO_UDINT(LEN(TTA.UpperLimit)), 
	pDest 			:= ADR(SendTelegram), 
	DestLen 		:= SIZEOF(SendTelegram), 
	WritePointer	:= mWritePointer);
	
F_AssembleByteStream(
	pSrc 			:= ADR(TTA.Sequence), 
	SrcLen 			:= INT_TO_UDINT(LEN(TTA.Sequence)), 
	pDest 			:= ADR(SendTelegram), 
	DestLen 		:= SIZEOF(SendTelegram), 
	WritePointer	:= mWritePointer);
	
F_AssembleByteStream(
	pSrc 			:= ADR(TTA.SubSequence), 
	SrcLen 			:= INT_TO_UDINT(LEN(TTA.SubSequence)), 
	pDest 			:= ADR(SendTelegram), 
	DestLen 		:= SIZEOF(SendTelegram), 
	WritePointer	:= mWritePointer);

F_AssembleByteStream(
	pSrc 			:= ADR(TTA.SequenceSize), 
	SrcLen 			:= INT_TO_UDINT(LEN(TTA.SequenceSize)), 
	pDest 			:= ADR(SendTelegram), 
	DestLen 		:= SIZEOF(SendTelegram), 
	WritePointer	:= mWritePointer);	

F_AssembleByteStream(
	pSrc 			:= ADR(TTA.GroupID), 
	SrcLen 			:= INT_TO_UDINT(LEN(TTA.GroupID)), 
	pDest 			:= ADR(SendTelegram), 
	DestLen 		:= SIZEOF(SendTelegram), 
	WritePointer	:= mWritePointer);	

F_AssembleByteStream(
	pSrc 			:= ADR(TTA.GroupSize), 
	SrcLen 			:= INT_TO_UDINT(LEN(TTA.GroupSize)), 
	pDest 			:= ADR(SendTelegram), 
	DestLen 		:= SIZEOF(SendTelegram), 
	WritePointer	:= mWritePointer);	

F_AssembleByteStream(
	pSrc 			:= ADR(TTA.DestinationSlot), 
	SrcLen 			:= INT_TO_UDINT(LEN(TTA.DestinationSlot)), 
	pDest 			:= ADR(SendTelegram), 
	DestLen 		:= SIZEOF(SendTelegram), 
	WritePointer	:= mWritePointer);	
	
F_AssembleByteStream(
	pSrc 			:= ADR(TTA.NumberOfDestinations), 
	SrcLen 			:= INT_TO_UDINT(LEN(TTA.NumberOfDestinations)), 
	pDest 			:= ADR(SendTelegram), 
	DestLen 		:= SIZEOF(SendTelegram), 
	WritePointer	:= mWritePointer);	

FOR mIdx := 1 TO TU_DataTable[mTU_DataIndex].DataSet.NumberOfDest DO
	F_AssembleByteStream(
		pSrc 			:= ADR(TTA.Destination[mIdx]), 
		SrcLen 			:= INT_TO_UDINT(LEN(TTA.Destination[mIdx])), 
		pDest 			:= ADR(SendTelegram), 
		DestLen 		:= SIZEOF(SendTelegram), 
		WritePointer	:= mWritePointer);	
END_FOR	

M_SendTTA := fbMFCS_SIS_Sub.M_SendAppData(pData := ADR(SendTelegram), DataLen := mWritePointer);
END_METHOD

END_FUNCTION_BLOCK

// ---- 20_Product/10_BCF/11_Conv/11_Com/13_Sub-Sub/FB_STI_SendTU_Trigger_6_0.TcPOU
FUNCTION_BLOCK FB_STI_SendTU_Trigger_6_0
(**************************************************************************************
 * 	Application		:	BoxControl Framework
 *	Revision		:	$Revision: 404529 $
 *	Revision date	:	$Date: 2018-04-23 08:21:38 +0200 (Mo., 23 Apr 2018) $
 *	Last changed by	:	$Author: b7bolm $
 *	URL				:	$URL: http://almscdc.swisslog.com/repo/SWPD/Development/BoxControlFramework/20_Release/trunk/01_Software/BCF/BCF/JumpStart/20_Product/10_App/11_Com/10_Lib/10_Conv/13_Sub-Sub/FB_STI_SendTU_Trigger_6_0.TcPOU $
 *
 *	Purpose			:	Triggers sending TTA over FB_STI_SendReceiveTU_Data to other SubSystem
 *
 * ------------------------------------------------------------------------------------
 *	Copyright Swisslog [IP AG], Switzerland. All rights reserved.
 * 
 * ------------------------------------------------------------------------------------
 *	
 * 	Revision History: 
 *
 *  VERSION DATE         INITIALS     DESCRIPTION
 *  0.0     DD.MM.YYYY   (name)       (explain customized modifications)
 *
 **************************************************************************************)
VAR_INPUT
	TriggerSendTU_Data		: BOOL; // TU-Data will be sent by trigger input (ignores zone occupied)
	SendTU_DataOccupied		: BOOL; // TU-Data will be sent when zone gets occupied
	eAssignedFunction		: E_FunctionNumber; // Assigned function number
	AssignedZone			: INT; // Assigned zone number
	DeleteTU_Data			: BOOL; // TU-data will be deleted after sending TTA
END_VAR
VAR_IN_OUT
	fbSendReceiveTU_Data	: FB_STI_SendReceiveTU_Data_6_0;
END_VAR
VAR
	Init					: BOOL := FALSE; // Instance is initialized
	fbDebugMsg				: FB_DebugMsg; // Debug instance
	DebugMsg				: T_MAXSTRING; // Debug msg
	State					: INT; // TTA sending state
	ZoneData 				: ST_ZoneData; // Zone data
	TU_DataIndex			: DINT; // TU data index
END_VAR

// Get zone data
ZoneData := F_GetZoneData(eFunctionNumber := eAssignedFunction, ZoneNumber := AssignedZone);

CASE State OF	
	
	0: // Init
		State := 10;
	
	
	10: // Wait for trigger
		IF TriggerSendTU_Data OR SendTU_DataOccupied AND ZoneData.TransportControlData.Occupied THEN
			TU_DataIndex := ZoneData.TransportControlData.TU_DataIndex;
			State := 20;
		END_IF
	
	
	20: // Send TU-data
		// TU-data present
		IF TU_DataIndex <> 0 THEN
			IF fbSendReceiveTU_Data.M_SendTTA(TU_DataIndex) THEN
				// Check if TU-data must be deleted
				IF DeleteTU_Data THEN
					State := 30;
				ELSE
					State := 40;
				END_IF
			END_IF
			
		// No TU-data to send
		ELSE
			State := 40;
		END_IF
		
		
	30: // Delete TU-data
		// debug message: '11-000-0000-00-0,  send TU_DataIndex deleted, position = 99-999-9999-99-9,  TU_DataIndex = 5,  TuID = 000012345,  AssignmentID = 999999999'
		DebugMsg := '';
		DebugMsg := CONCAT(DebugMsg, F_AddDividerToSisString(SubsystemRegistry.SubsystemName));
		DebugMsg := CONCAT(DebugMsg, ',  send TU_DataIndex deleted');
		DebugMsg := CONCAT(DebugMsg, DebugTextBlocks.POSITION);
		DebugMsg := CONCAT(DebugMsg, F_GetFunctionName(eFunctionNumber:= eAssignedFunction, ZoneNumber:= 0));
		DebugMsg := CONCAT(DebugMsg, F_CreateTU_DataString(TU_DataIndex:= TU_DataIndex));
		fbDebugMsg.M_SendInfoMsg(DebugMsg);
		F_DeleteTU_Data(
			TU_DataIndex 	:= TU_DataIndex,
			NoTTC			:= TRUE);
		
		State := 40;
		

	40: // Wait until trigger is reset or zone is free
		IF NOT TriggerSendTU_Data OR SendTU_DataOccupied AND NOT ZoneData.TransportControlData.Occupied THEN
			State := 10;
		END_IF	
	
END_CASE

END_FUNCTION_BLOCK

// ---- 20_Product/10_BCF/11_Conv/11_Com/13_Sub-Sub/FB_STI_SendTU_Trigger_6_1.TcPOU
FUNCTION_BLOCK FB_STI_SendTU_Trigger_6_1
(**************************************************************************************
 * 	Application		:	BoxControl Framework
 *	Revision		:	$Revision: 404529 $
 *	Revision date	:	$Date: 2018-04-23 08:21:38 +0200 (Mo., 23 Apr 2018) $
 *	Last changed by	:	$Author: b7bolm $
 *	URL				:	$URL: http://almscdc.swisslog.com/repo/SWPD/Development/BoxControlFramework/20_Release/trunk/01_Software/BCF/BCF/JumpStart/20_Product/10_App/11_Com/10_Lib/10_Conv/13_Sub-Sub/FB_STI_SendTU_Trigger_6_1.TcPOU $
 *
 *	Purpose			:	Triggers sending TTA over FB_STI_SendReceiveTU_Data to other SubSystem
 *
 * ------------------------------------------------------------------------------------
 *	Copyright Swisslog [IP AG], Switzerland. All rights reserved.
 * 
 * ------------------------------------------------------------------------------------
 *	
 * 	Revision History: 
 *
 *  VERSION DATE         INITIALS     DESCRIPTION
 *  0.0     DD.MM.YYYY   (name)       (explain customized modifications)
 *
 **************************************************************************************)
VAR_INPUT
	TriggerSendTU_Data		: BOOL; // TU-Data will be sent by trigger input (ignores zone occupied)
	SendTU_DataOccupied		: BOOL; // TU-Data will be sent when zone gets occupied
	eAssignedFunction		: E_FunctionNumber; // Assigned function number
	AssignedZone			: INT; // Assigned zone number
	DeleteTU_Data			: BOOL; // TU-data will be deleted after sending TTA
END_VAR
VAR_IN_OUT
	fbSendReceiveTU_Data	: FB_STI_SendReceiveTU_Data_6_1;
END_VAR
VAR
	Init					: BOOL := FALSE; // Instance is initialized
	fbDebugMsg				: FB_DebugMsg; // Debug instance
	DebugMsg				: T_MAXSTRING; // Debug msg
	State					: INT; // TTA sending state
	ZoneData 				: ST_ZoneData; // Zone data
	TU_DataIndex			: DINT; // TU data index
END_VAR

// Get zone data
ZoneData := F_GetZoneData(eFunctionNumber := eAssignedFunction, ZoneNumber := AssignedZone);

CASE State OF	
	
	0: // Init
		State := 10;
	
	
	10: // Wait for trigger
		IF TriggerSendTU_Data OR SendTU_DataOccupied AND ZoneData.TransportControlData.Occupied THEN
			TU_DataIndex := ZoneData.TransportControlData.TU_DataIndex;
			State := 20;
		END_IF
	
	
	20: // Send TU-data
		// TU-data present
		IF TU_DataIndex <> 0 THEN
			IF fbSendReceiveTU_Data.M_SendTTA(TU_DataIndex) THEN
				// Check if TU-data must be deleted
				IF DeleteTU_Data THEN
					State := 30;
				ELSE
					State := 40;
				END_IF
			END_IF
			
		// No TU-data to send
		ELSE
			State := 40;
		END_IF
		
		
	30: // Delete TU-data
		// debug message: '11-000-0000-00-0,  send TU_DataIndex deleted, position = 99-999-9999-99-9,  TU_DataIndex = 5,  TuID = 000012345,  AssignmentID = 999999999'
		DebugMsg := '';
		DebugMsg := CONCAT(DebugMsg, F_AddDividerToSisString(SubsystemRegistry.SubsystemName));
		DebugMsg := CONCAT(DebugMsg, ',  send TU_DataIndex deleted');
		DebugMsg := CONCAT(DebugMsg, DebugTextBlocks.POSITION);
		DebugMsg := CONCAT(DebugMsg, F_GetFunctionName(eFunctionNumber:= eAssignedFunction, ZoneNumber:= 0));
		DebugMsg := CONCAT(DebugMsg, F_CreateTU_DataString(TU_DataIndex:= TU_DataIndex));
		fbDebugMsg.M_SendInfoMsg(DebugMsg);
		F_DeleteTU_Data(
			TU_DataIndex 	:= TU_DataIndex,
			NoTTC			:= TRUE);
		
		State := 40;
		

	40: // Wait until trigger is reset or zone is free
		IF NOT TriggerSendTU_Data OR SendTU_DataOccupied AND NOT ZoneData.TransportControlData.Occupied THEN
			State := 10;
		END_IF	
	
END_CASE

END_FUNCTION_BLOCK

// ---- 20_Product/10_BCF/11_Conv/12_E_Functions/09_Emulation/FB_FunctionConvEmulation.TcPOU
FUNCTION_BLOCK FB_FunctionConvEmulation EXTENDS FB_BaseObjectEmulation
(**************************************************************************************
 * 	Application		:	BoxControl Framework
 *	Revision		:	$Revision: 461869 $
 *	Revision date	:	$Date: 2020-09-25 14:40:24 +0200 (fre, 25 sep 2020) $
 *	Last changed by	:	$Author: d7mangc $
 *	URL				:	$URL: http://almscdc.swisslog.com/repo/SWPD/Development/BoxControlFramework/20_Release/tags/R1.12.0/01_Software/BCF/BCF/JumpStart/20_Product/10_BCF/11_Conv/12_E_Functions/09_Emulation/FB_FunctionConvEmulation.TcPOU $
 *
 *	Purpose			:	Base emulation function.
 *
 * ------------------------------------------------------------------------------------
 *	Copyright Swisslog [IP AG], Switzerland. All rights reserved.
 * 
 * --------------------------- ---------------------------------------------------------
 *	
 * 	Revision History: 
 *
 * 	VERSION			DATE			INITIALS			DESCRIPTION
 *	0.1				01.01.2001		swl					Example
 *
 **************************************************************************************)
VAR_INPUT
	eFunctionNumber					: E_FunctionNumber; // Function number
END_VAR

VAR
	FunctionBase					: ST_FunctionBaseEmulation; // Collecting variables used by framework
	Idx								: INT; // Iterator
END_VAR

VAR PERSISTENT
	ITC								: ST_ITC_FunctionEmulation; // ITC Emulation	
	FunctionData					: ST_FunctionDataEmulation; // Function data emulation
	ZoneData						: ARRAY[1..NUMBER_OF_ZONES_PER_FUNCTION] OF ST_ZoneDataEmulation; // Zone data
END_VAR

;

ACTION A_ExternalSTI:
(**************************************************************************************
 * 	NAME		A_ExternalSTI
 * 	FUNCTION	External Subsystem transport interface
 **************************************************************************************)


(**************************************************************************************
   External Subsystem transport interfaces
***************************************************************************************)
FOR Idx := 1 TO NUMBER_OF_STI DO
	// Is an external Subsystem transport interface configured
	IF FunctionBase.rSettingsFunctionReal.eExternalSTI_FunctionNumber[Idx] > E_FunctionNumber.F_BEGIN_EXTERN_FUNCTION AND
	   FunctionBase.rSettingsFunctionReal.eExternalSTI_FunctionNumber[Idx] < E_FunctionNumber.F_END_EXTERN_FUNCTION THEN
	   
		// When interface is valid
		IF __QUERYINTERFACE(fbSTI_ChannelsEmulation[FunctionBase.rSettingsFunctionReal.eExternalSTI_FunctionNumber[Idx]].Instance,FunctionBase.STI_Instance) THEN
			// Call external inbound interface
			fbSTI_ChannelsEmulation[FunctionBase.rSettingsFunctionReal.eExternalSTI_FunctionNumber[Idx]].Instance.M_CallInterface();
		END_IF
	END_IF
END_FOR
END_ACTION

METHOD PROTECTED M_GetNextTransportData : REFERENCE TO ST_TransportDataEmulation
(**************************************************************************************
 * 	Application		:	BoxControl Framework
 *	Revision		:	$Revision: 461869 $
 *	Revision date	:	$Date: 2020-09-25 14:40:24 +0200 (fre, 25 sep 2020) $
 *	Last changed by	:	$Author: d7mangc $
 *	URL				:	$URL: http://almscdc.swisslog.com/repo/SWPD/Development/BoxControlFramework/20_Release/tags/R1.12.0/01_Software/BCF/BCF/JumpStart/20_Product/10_BCF/11_Conv/12_E_Functions/09_Emulation/FB_FunctionConvEmulation.TcPOU $
 *
 *	Purpose			:	Get transport data for next zone
 *
 * ------------------------------------------------------------------------------------
 *	Copyright Swisslog [IP AG], Switzerland. All rights reserved.
 * 
 * ------------------------------------------------------------------------------------
 *	
 * 	Revision History: 
 *
 * 	VERSION			DATE			INITIALS			DESCRIPTION
 *	0.1				01.01.2001		swl					Example
 *
 **************************************************************************************)
VAR_INPUT
	mZoneNumber : INT; // Number of the zone
END_VAR

VAR
	meFunctionNumber : E_FunctionNumber;
END_VAR
(*
Initialize
Reference points initialy to an empty struct, to ensure
always a valid reference, even no decision could be made.
*)

FunctionBase.TransportDataEmpty.eFunctionNumber := E_FunctionNumber.F_BEGIN_FUNCTION;
FunctionBase.TransportDataEmpty.ZoneNumber := 0;
FunctionBase.TransportDataEmpty.rTransportControlData REF= FunctionBase.TransportControlDataEmptyEmulation;
FunctionBase.TransportDataEmpty.rSettings REF= FunctionBase.ZoneSettingsEmpty;
FunctionBase.TransportDataEmpty.rRealObjTrspControlData REF= FunctionBase.TransportControlDataEmpty;
M_GetNextTransportData REF= FunctionBase.TransportDataEmpty;

// If flow direction is forward
IF NOT FunctionBase.rSettingsFunctionReal.FlowDirectionREV THEN
	// If is it the last zone within the function 
	IF mZoneNumber = FunctionBase.rSettingsFunctionReal.NumberOfZones THEN
		// If the function number is valid
		IF FunctionBase.rFunctionInterfaceReal.In.eNextFunctionNumber > F_BEGIN_FUNCTION AND
           FunctionBase.rFunctionInterfaceReal.In.eNextFunctionNumber < F_END_FUNCTION THEN

			meFunctionNumber := FunctionBase.rFunctionInterfaceReal.In.eNextFunctionNumber;
			
			// If the reference is valid and the real function is initialized
			IF __ISVALIDREF(FunctionRegistryEmulation[meFunctionNumber].rFunction) AND
			   F_IsFunctionInitialized(meFunctionNumber) THEN 
				// Return adjacent transport data of the adjacent function
				M_GetNextTransportData REF= FunctionRegistryEmulation[meFunctionNumber].rFunction.
											M_GetTransportData(meFunctionNumber := FunctionBase.rSettingsFunctionReal.eFunctionNumber);
			END_IF

		// If the function number points to an external interface
		ELSIF FunctionBase.rFunctionInterfaceReal.In.eNextFunctionNumber > E_FunctionNumber.F_BEGIN_EXTERN_FUNCTION AND
			  FunctionBase.rFunctionInterfaceReal.In.eNextFunctionNumber < E_FunctionNumber.F_END_EXTERN_FUNCTION THEN
			
			// If the reference is valid and the real function is initialized
			IF __QUERYINTERFACE(fbSTI_ChannelsEmulation[FunctionBase.rFunctionInterfaceReal.In.eNextFunctionNumber].Instance,FunctionBase.STI_Instance) THEN
				// Return adjacent transport data of the adjacent function
				M_GetNextTransportData REF= fbSTI_ChannelsEmulation[FunctionBase.rFunctionInterfaceReal.In.eNextFunctionNumber].Instance.M_GetTransportData();
			END_IF
		END_IF
	ELSE
		// Return trasnport data of the previous function internal zone
		FunctionBase.NextTransportData.eFunctionNumber := FunctionBase.rSettingsFunctionReal.eFunctionNumber;
		FunctionBase.NextTransportData.ZoneNumber := mZoneNumber +1;
		FunctionBase.NextTransportData.rTransportControlData REF= ZoneData[mZoneNumber +1].TransportControlData;
		FunctionBase.NextTransportData.rSettings REF= FunctionBase.rSettingsFunctionReal.Zone[mZoneNumber +1];
		FunctionBase.NextTransportData.rRealObjTrspControlData REF= FunctionBase.rZoneDataReal[mZoneNumber +1].TransportControlData;
		M_GetNextTransportData REF= FunctionBase.NextTransportData;
	END_IF

// Flow direction is reverse
ELSE
	// If is it the first zone within the function 
	IF mZoneNumber = 1 THEN
		// If then function number is valid
		IF FunctionBase.rFunctionInterfaceReal.In.eNextFunctionNumber > F_BEGIN_FUNCTION AND
           FunctionBase.rFunctionInterfaceReal.In.eNextFunctionNumber < F_END_FUNCTION THEN
		   
			meFunctionNumber := FunctionBase.rFunctionInterfaceReal.In.eNextFunctionNumber;
			
			// If the reference is valid and the real function is initialized
			IF __ISVALIDREF(FunctionRegistryEmulation[meFunctionNumber].rFunction) AND
			   F_IsFunctionInitialized(meFunctionNumber) THEN
				// Return adjacent transport data of the adjacent function
				M_GetNextTransportData REF= FunctionRegistryEmulation[meFunctionNumber].rFunction.
											M_GetTransportData(meFunctionNumber := FunctionBase.rSettingsFunctionReal.eFunctionNumber);	
			END_IF

		// If the function number points to an external interface
		ELSIF FunctionBase.rFunctionInterfaceReal.In.eNextFunctionNumber > E_FunctionNumber.F_BEGIN_EXTERN_FUNCTION AND
			  FunctionBase.rFunctionInterfaceReal.In.eNextFunctionNumber < E_FunctionNumber.F_END_EXTERN_FUNCTION THEN
			  
			// If the reference is valid and the real function is initialized
			IF __QUERYINTERFACE(fbSTI_ChannelsEmulation[FunctionBase.rFunctionInterfaceReal.In.eNextFunctionNumber].Instance,FunctionBase.STI_Instance) THEN
				// Return adjacent transport data of the adjacent function
				M_GetNextTransportData REF= fbSTI_ChannelsEmulation[FunctionBase.rFunctionInterfaceReal.In.eNextFunctionNumber].Instance.M_GetTransportData();
			END_IF
		END_IF
	ELSE
		// Return trasnport data of the previous function internal zone
		FunctionBase.NextTransportData.eFunctionNumber := FunctionBase.rSettingsFunctionReal.eFunctionNumber;
		FunctionBase.NextTransportData.ZoneNumber := mZoneNumber -1;	
		FunctionBase.NextTransportData.rTransportControlData REF= ZoneData[mZoneNumber -1].TransportControlData;
		FunctionBase.NextTransportData.rSettings REF= FunctionBase.rSettingsFunctionReal.Zone[mZoneNumber -1];
		FunctionBase.NextTransportData.rRealObjTrspControlData REF= FunctionBase.rZoneDataReal[mZoneNumber -1].TransportControlData;
		M_GetNextTransportData REF= FunctionBase.NextTransportData;
	END_IF
END_IF
END_METHOD

METHOD PROTECTED M_GetPreviousTransportData : REFERENCE TO ST_TransportDataEmulation
(**************************************************************************************
 * 	Application		:	BoxControl Framework
 *	Revision		:	$Revision: 461869 $
 *	Revision date	:	$Date: 2020-09-25 14:40:24 +0200 (fre, 25 sep 2020) $
 *	Last changed by	:	$Author: d7mangc $
 *	URL				:	$URL: http://almscdc.swisslog.com/repo/SWPD/Development/BoxControlFramework/20_Release/tags/R1.12.0/01_Software/BCF/BCF/JumpStart/20_Product/10_BCF/11_Conv/12_E_Functions/09_Emulation/FB_FunctionConvEmulation.TcPOU $
 *
 *	Purpose			:	Get transport data from previous zone
 *
 * ------------------------------------------------------------------------------------
 *	Copyright Swisslog [IP AG], Switzerland. All rights reserved.
 * 
 * ------------------------------------------------------------------------------------
 *	
 * 	Revision History: 
 *
 * 	VERSION			DATE			INITIALS			DESCRIPTION
 *	0.1				01.01.2001		swl					Example
 *
 **************************************************************************************)
VAR_INPUT
	mZoneNumber : INT; // Number of the zone
END_VAR

VAR
	meFunctionNumber : E_FunctionNumber;
END_VAR
(*
Initialize
Reference points initialy to an empty struct, to ensure
always a valid reference, even no decision could be made.
*)

FunctionBase.TransportDataEmpty.eFunctionNumber := E_FunctionNumber.F_BEGIN_FUNCTION;
FunctionBase.TransportDataEmpty.ZoneNumber := 0;
FunctionBase.TransportDataEmpty.rTransportControlData REF= FunctionBase.TransportControlDataEmptyEmulation;
FunctionBase.TransportDataEmpty.rSettings REF= FunctionBase.ZoneSettingsEmpty;
FunctionBase.TransportDataEmpty.rRealObjTrspControlData REF= FunctionBase.TransportControlDataEmpty;
M_GetPreviousTransportData REF= FunctionBase.TransportDataEmpty;

// If flow direction is forward
IF NOT FunctionBase.rSettingsFunctionReal.FlowDirectionREV THEN 
	// If is it the first zone within the function
	IF mZoneNumber = 1 THEN
		// If the function number is valid
		IF FunctionBase.rFunctionInterfaceReal.In.ePrevFunctionNumber > F_BEGIN_FUNCTION AND
           FunctionBase.rFunctionInterfaceReal.In.ePrevFunctionNumber < F_END_FUNCTION THEN
		   
		   meFunctionNumber := FunctionBase.rFunctionInterfaceReal.In.ePrevFunctionNumber;
		   
			// If the reference is valid and the real function is initialized
			IF __ISVALIDREF(FunctionRegistryEmulation[meFunctionNumber].rFunction) AND
			   F_IsFunctionInitialized(meFunctionNumber) THEN
				// Return adjacent transport data of the adjacent function
				M_GetPreviousTransportData REF= FunctionRegistryEmulation[meFunctionNumber].rFunction.M_GetTransportData(
													meFunctionNumber :=FunctionBase.rSettingsFunctionReal.eFunctionNumber);
			END_IF

		// If the function number points to an external interface
		ELSIF FunctionBase.rFunctionInterfaceReal.In.ePrevFunctionNumber > E_FunctionNumber.F_BEGIN_EXTERN_FUNCTION AND
			  FunctionBase.rFunctionInterfaceReal.In.ePrevFunctionNumber < E_FunctionNumber.F_END_EXTERN_FUNCTION THEN

			// If the reference is valid and the real function is initialized
			IF __QUERYINTERFACE(fbSTI_ChannelsEmulation[FunctionBase.rFunctionInterfaceReal.In.ePrevFunctionNumber].Instance,FunctionBase.STI_Instance) THEN
				// If the reference is valid and the real function is initialized
				M_GetPreviousTransportData REF= fbSTI_ChannelsEmulation[FunctionBase.rFunctionInterfaceReal.In.ePrevFunctionNumber].Instance.M_GetTransportData();
			END_IF
		END_IF
	ELSE
		// Return trasnport data of the previous function internal zone
		FunctionBase.PrevTransportData.eFunctionNumber := FunctionBase.rSettingsFunctionReal.eFunctionNumber;
		FunctionBase.PrevTransportData.ZoneNumber := mZoneNumber -1;	
		FunctionBase.PrevTransportData.rTransportControlData REF= ZoneData[mZoneNumber -1].TransportControlData;
		FunctionBase.PrevTransportData.rSettings REF= FunctionBase.rSettingsFunctionReal.Zone[mZoneNumber -1];
		FunctionBase.PrevTransportData.rRealObjTrspControlData REF= FunctionBase.rZoneDataReal[mZoneNumber -1].TransportControlData;
		M_GetPreviousTransportData REF= FunctionBase.PrevTransportData;
	END_IF

// Flow direction is reverse
ELSE
	// If is it the last zone within the function
	IF mZoneNumber = FunctionBase.rSettingsFunctionReal.NumberOfZones THEN
		// If the function number is valid
		IF FunctionBase.rFunctionInterfaceReal.In.ePrevFunctionNumber > F_BEGIN_FUNCTION AND
           FunctionBase.rFunctionInterfaceReal.In.ePrevFunctionNumber < F_END_FUNCTION THEN
			
			meFunctionNumber := FunctionBase.rFunctionInterfaceReal.In.ePrevFunctionNumber;
		   
			// If the reference is valid and the real function is initialized
			IF __ISVALIDREF(FunctionRegistryEmulation[meFunctionNumber].rFunction) AND
			   F_IsFunctionInitialized(meFunctionNumber) THEN
				// Return adjacent transport data of the adjacent function
				M_GetPreviousTransportData REF= FunctionRegistryEmulation[meFunctionNumber].rFunction.M_GetTransportData(
													meFunctionNumber := FunctionBase.rSettingsFunctionReal.eFunctionNumber);
			END_IF

		// If the function number points to an external interface
		ELSIF FunctionBase.rFunctionInterfaceReal.In.ePrevFunctionNumber > E_FunctionNumber.F_BEGIN_EXTERN_FUNCTION AND
			  FunctionBase.rFunctionInterfaceReal.In.ePrevFunctionNumber < E_FunctionNumber.F_END_EXTERN_FUNCTION THEN
			  
			// If the reference is valid and the real function is initialized
			IF __QUERYINTERFACE(fbSTI_ChannelsEmulation[FunctionBase.rFunctionInterfaceReal.In.ePrevFunctionNumber].Instance,FunctionBase.STI_Instance) THEN
				// If the reference is valid and the real function is initialized
				M_GetPreviousTransportData REF= fbSTI_ChannelsEmulation[FunctionBase.rFunctionInterfaceReal.In.ePrevFunctionNumber].Instance.M_GetTransportData();
			END_IF
		END_IF
	ELSE
		// Return trasnport data of the previous function internal zone
		FunctionBase.PrevTransportData.eFunctionNumber := FunctionBase.rSettingsFunctionReal.eFunctionNumber;
		FunctionBase.PrevTransportData.ZoneNumber := mZoneNumber +1;	
		FunctionBase.PrevTransportData.rTransportControlData REF= ZoneData[mZoneNumber +1].TransportControlData;
		FunctionBase.PrevTransportData.rSettings REF= FunctionBase.rSettingsFunctionReal.Zone[mZoneNumber +1];
		FunctionBase.PrevTransportData.rRealObjTrspControlData REF= FunctionBase.rZoneDataReal[mZoneNumber +1].TransportControlData;
		M_GetPreviousTransportData REF= FunctionBase.PrevTransportData;
	END_IF
END_IF
END_METHOD

METHOD PROTECTED M_GetTransportControlParam : REFERENCE TO ST_TransportControlParam
(**************************************************************************************
 * 	Application		:	BoxControl Framework
 *	Revision		:	$Revision: 461869 $
 *	Revision date	:	$Date: 2020-09-25 14:40:24 +0200 (fre, 25 sep 2020) $
 *	Last changed by	:	$Author: d7mangc $
 *	URL				:	$URL: http://almscdc.swisslog.com/repo/SWPD/Development/BoxControlFramework/20_Release/tags/R1.12.0/01_Software/BCF/BCF/JumpStart/20_Product/10_BCF/11_Conv/12_E_Functions/09_Emulation/FB_FunctionConvEmulation.TcPOU $
 *
 *	Purpose			:	Get transport control parameter
 *
 * ------------------------------------------------------------------------------------
 *	Copyright Swisslog [IP AG], Switzerland. All rights reserved.
 * 
 * ------------------------------------------------------------------------------------
 *	
 * 	Revision History: 
 *
 * 	VERSION			DATE			INITIALS			DESCRIPTION
 *	0.1				01.01.2001		swl					Example
 *
 **************************************************************************************)
VAR_INPUT
	mZoneNumber 			: INT; // Number of the zone
END_VAR

// Return function number
FunctionBase.TransportControlParam.reFunctionNumber REF= FunctionBase.rSettingsFunctionReal.eFunctionNumber;
// Return function state
FunctionBase.TransportControlParam.rOperationState REF= FunctionBase.rFunctionDataReal.OperationState;
// Return zone number
FunctionBase.TransportControlParam.ZoneNumber := mZoneNumber;
// Return zone settings
FunctionBase.TransportControlParam.rSettings REF= FunctionBase.rSettingsFunctionReal.Zone[mZoneNumber];
// Return zone enable
FunctionBase.TransportControlParam.rZoneEnable REF= FunctionBase.rZoneInterfaceReal[mZoneNumber].In.Enable;
// Return external zone enable
FunctionBase.TransportControlParam.rExternalZoneEnable REF= FunctionBase.rZoneInterfaceReal[mZoneNumber].In.ZoneEnable;

M_GetTransportControlParam REF= FunctionBase.TransportControlParam;
END_METHOD

METHOD M_GetTransportData : REFERENCE TO ST_TransportDataEmulation;
(**************************************************************************************
 * 	Application		:	BoxControl Framework
 *	Revision		:	$Revision: 461869 $
 *	Revision date	:	$Date: 2020-09-25 14:40:24 +0200 (fre, 25 sep 2020) $
 *	Last changed by	:	$Author: d7mangc $
 *	URL				:	$URL: http://almscdc.swisslog.com/repo/SWPD/Development/BoxControlFramework/20_Release/tags/R1.12.0/01_Software/BCF/BCF/JumpStart/20_Product/10_BCF/11_Conv/12_E_Functions/09_Emulation/FB_FunctionConvEmulation.TcPOU $
 *
 *	Purpose			:	Get adjacent zone
 *
 * ------------------------------------------------------------------------------------
 *	Copyright Swisslog [IP AG], Switzerland. All rights reserved.
 * 
 * ------------------------------------------------------------------------------------
 *	
 * 	Revision History: 
 *
 * 	VERSION			DATE			INITIALS			DESCRIPTION
 *	0.1				01.01.2001		swl					Example
 *
 **************************************************************************************)
VAR_INPUT
	meFunctionNumber : E_FunctionNumber; // Own element function number
END_VAR
(*
Initialize
Reference points initialy to an empty struct, to ensure
always a valid reference, even no decision could be made.
*)
FunctionBase.TransportDataEmpty.eFunctionNumber := E_FunctionNumber.F_BEGIN_FUNCTION;
FunctionBase.TransportDataEmpty.ZoneNumber := 0;
FunctionBase.TransportDataEmpty.rTransportControlData REF= FunctionBase.TransportControlDataEmptyEmulation;
FunctionBase.TransportDataEmpty.rSettings REF= FunctionBase.ZoneSettingsEmpty;
FunctionBase.TransportDataEmpty.rRealObjTrspControlData REF= FunctionBase.TransportControlDataEmpty;
M_GetTransportData REF= FunctionBase.TransportDataEmpty;

// If the function number is valid and function is initialized
IF meFunctionNumber > F_BEGIN_FUNCTION AND FunctionData.Init THEN
	// If the requesting function is the previous function
	IF meFunctionNumber = FunctionBase.rFunctionInterfaceReal.In.ePrevFunctionNumber THEN
		
		// If the flow direction is forward
		IF NOT FunctionBase.rSettingsFunctionReal.FlowDirectionREV THEN
			// Return the transport data of the first zone
			FunctionBase.TransportData.eFunctionNumber := FunctionBase.rSettingsFunctionReal.eFunctionNumber;
			FunctionBase.TransportData.ZoneNumber := 1;
			FunctionBase.TransportData.rSettings REF= FunctionBase.rSettingsFunctionReal.Zone[1];
			FunctionBase.TransportData.rTransportControlData REF= ZoneData[1].TransportControlData;
			FunctionBase.TransportData.rRealObjTrspControlData REF= FunctionBase.rZoneDataReal[1].TransportControlData;
			M_GetTransportData REF= FunctionBase.TransportData;
		ELSE
			// If the zone number is valid
			IF FunctionBase.rSettingsFunctionReal.NumberOfZones <> 0 THEN
				// Return the transport data of the last zone
				FunctionBase.TransportData.eFunctionNumber := FunctionBase.rSettingsFunctionReal.eFunctionNumber;
				FunctionBase.TransportData.ZoneNumber := FunctionBase.rSettingsFunctionReal.NumberOfZones;
				FunctionBase.TransportData.rSettings REF= FunctionBase.rSettingsFunctionReal.Zone[FunctionBase.rSettingsFunctionReal.NumberOfZones];
				FunctionBase.TransportData.rTransportControlData REF= ZoneData[FunctionBase.rSettingsFunctionReal.NumberOfZones].TransportControlData;
				FunctionBase.TransportData.rRealObjTrspControlData REF= FunctionBase.rZoneDataReal[FunctionBase.rSettingsFunctionReal.NumberOfZones].TransportControlData;	
				M_GetTransportData REF= FunctionBase.TransportData;	
			END_IF	
		END_IF
	
	// If the requesting function is the next function
	ELSIF meFunctionNumber = FunctionBase.rFunctionInterfaceReal.In.eNextFunctionNumber THEN
		
		// If the flow direction is forward
		IF NOT FunctionBase.rSettingsFunctionReal.FlowDirectionREV THEN
			// If the zone number is valid
			IF FunctionBase.rSettingsFunctionReal.NumberOfZones <> 0 THEN
				// Return the transport data of the last zone
				FunctionBase.TransportData.eFunctionNumber := FunctionBase.rSettingsFunctionReal.eFunctionNumber;
				FunctionBase.TransportData.ZoneNumber := FunctionBase.rSettingsFunctionReal.NumberOfZones;
				FunctionBase.TransportData.rSettings REF= FunctionBase.rSettingsFunctionReal.Zone[FunctionBase.rSettingsFunctionReal.NumberOfZones];
				FunctionBase.TransportData.rTransportControlData REF= ZoneData[FunctionBase.rSettingsFunctionReal.NumberOfZones].TransportControlData;
				FunctionBase.TransportData.rRealObjTrspControlData REF= FunctionBase.rZoneDataReal[FunctionBase.rSettingsFunctionReal.NumberOfZones].TransportControlData;	
				M_GetTransportData REF= FunctionBase.TransportData;	
			END_IF
		ELSE
			// Return the transport data of the first zone
			FunctionBase.TransportData.eFunctionNumber := FunctionBase.rSettingsFunctionReal.eFunctionNumber;
			FunctionBase.TransportData.ZoneNumber := 1;
			FunctionBase.TransportData.rSettings REF= FunctionBase.rSettingsFunctionReal.Zone[1];
			FunctionBase.TransportData.rTransportControlData REF= ZoneData[1].TransportControlData;
			FunctionBase.TransportData.rRealObjTrspControlData REF= FunctionBase.rZoneDataReal[1].TransportControlData;		
			M_GetTransportData REF= FunctionBase.TransportData;	
		END_IF
	END_IF
END_IF
END_METHOD

METHOD M_GetTU_PresentState : BOOL
(**************************************************************************************
 * 	Application		:	BoxControl Framework
 *	Revision		:	$Revision: 461869 $
 *	Revision date	:	$Date: 2020-09-25 14:40:24 +0200 (fre, 25 sep 2020) $
 *	Last changed by	:	$Author: d7mangc $
 *	URL				:	$URL: http://almscdc.swisslog.com/repo/SWPD/Development/BoxControlFramework/20_Release/tags/R1.12.0/01_Software/BCF/BCF/JumpStart/20_Product/10_BCF/11_Conv/12_E_Functions/09_Emulation/FB_FunctionConvEmulation.TcPOU $
 *
 *	Purpose			:	Base get TU present state, needs to be overriden from inheritance object
 *
 * ------------------------------------------------------------------------------------
 *	Copyright Swisslog [IP AG], Switzerland. All rights reserved.
 * 
 * ------------------------------------------------------------------------------------
 *	
 * 	Revision History: 
 *
 * 	VERSION			DATE			INITIALS			DESCRIPTION
 *	0.1				01.01.2001		swl					Example
 *
 **************************************************************************************)
VAR_INPUT
	mZone	 : INT; // Zone number
	mPosition : UINT; // Position [mm]
END_VAR
VAR_OUTPUT
	mTU_DataIndex : DINT;
END_VAR
;
END_METHOD

METHOD PRIVATE M_ITC_ATQ : BOOL
VAR_INPUT
	meChannelSrc		: E_MFCS_CHANNEL; // Number of the source 
	mpData				: PVOID; // Data  pointer 
	mLen				: UDINT; // Data length
END_VAR
// Map data
F_BlockCopy(
	pSrc:= mpData, 
	LenSrc:= mLen, 
	pDest:= ADR(FunctionBase.Data), 
	LenDest:= SIZEOF(FunctionBase.Data));
	
// If a data index is available
IF FunctionBase.Data.TU_DataIndex > 0 THEN
	// If a valid zone number is ready
	IF FunctionBase.Data.ZoneNumber > 0 THEN
		// Send "Add TU" request to zone
		ZoneData[FunctionBase.Data.ZoneNumber].ITC.Commands.AddTU := TRUE;
		ZoneData[FunctionBase.Data.ZoneNumber].ITC.Commands.TU_DataIndexToAdd := FunctionBase.Data.TU_DataIndex;
	ELSE
		// Invalid zone number
		DebugMsg := 'ADD_TU_DATA - No valid ZoneNumber, request rejected';
		fbDebugMsg.M_SendErrorMsg(DebugMsg);
	END_IF
ELSE
	// Invalid TU index
	DebugMsg := 'ADD_TU_DATA - No valid TU index, request rejected';
	fbDebugMsg.M_SendErrorMsg(DebugMsg);
END_IF
END_METHOD

METHOD PRIVATE M_ITC_ERQ : BOOL
(**************************************************************************************
 * 	Application		:	BoxControl Framework
 *	Revision		:	$Revision: 461869 $
 *	Revision date	:	$Date: 2020-09-25 14:40:24 +0200 (fre, 25 sep 2020) $
 *	Last changed by	:	$Author: d7mangc $
 *	URL				:	$URL: http://almscdc.swisslog.com/repo/SWPD/Development/BoxControlFramework/20_Release/tags/R1.12.0/01_Software/BCF/BCF/JumpStart/20_Product/10_BCF/11_Conv/12_E_Functions/09_Emulation/FB_FunctionConvEmulation.TcPOU $
 *
 *	Purpose			:	Add ERQ
 *
 * ------------------------------------------------------------------------------------
 *	Copyright Swisslog [IP AG], Switzerland. All rights reserved.
 * 
 * ------------------------------------------------------------------------------------
 *	
 * 	Revision History: 
 *
 * 	VERSION			DATE			INITIALS			DESCRIPTION
 *	0.1				01.01.2001		swl					Example
 *
 **************************************************************************************)
VAR_INPUT
	meChannelSrc		: E_MFCS_CHANNEL; // Number of the source 
	mpData				: PVOID; // Data  pointer 
	mLen				: UDINT; // Data length
END_VAR
// Map data
F_BlockCopy(
	pSrc:= mpData, 
	LenSrc:= mLen, 
	pDest:= ADR(FunctionBase.ERQ), 
	LenDest:= SIZEOF(FunctionBase.ERQ));		
	
FunctionBase.Position := F_SearchFunctionPosition(Position := FunctionBase.ERQ.Position);

// If request goes to function
IF FunctionBase.Position.ZoneNumber = 0 THEN
	// Send "Error" request to zone
	ITC.FunctionITC.Commands.Error := FunctionBase.ERQ.Code = 0;
	ITC.FunctionITC.Commands.ErrorCode := FunctionBase.ERQ.ErrorCode;
// If request has a zonenumber
ELSIF FunctionBase.Position.ZoneNumber > 0 THEN
	// Send "Error" request to zone
	ZoneData[FunctionBase.Position.ZoneNumber].ITC.Commands.Error := FunctionBase.ERQ.Code = 0;
	ZoneData[FunctionBase.Position.ZoneNumber].ITC.Commands.ErrorCode := FunctionBase.ERQ.ErrorCode;
ELSE
	// Invalid zone number
	DebugMsg := 'MODIFY_EMULATION_ERROR - No valid ZoneNumber, request rejected';
	fbDebugMsg.M_SendErrorMsg(DebugMsg);
END_IF
END_METHOD

METHOD M_ITC_ProcessMsg : BOOL
VAR_INPUT
	meChannelSrc		: E_MFCS_CHANNEL; // Number of the source 
	mMsgType			: INT; // Message type
	mpData				: PVOID; // Data  pointer 
	mLen				: UDINT; // Data length
END_VAR

// Initialize
M_ITC_ProcessMsg := TRUE;

// Validate inputs
IF mpData > 0 AND
   mLen > 0 THEN
	// map enum
	FunctionBase.eMsgType := mMsgType;

	// Validate message type
	CASE FunctionBase.eMsgType OF

		(*******************************************************************************
		  No Message
		********************************************************************************)
		E_ITC_MsgTypeConv.NO_MESSAGE_TYPE:
			// Empty message received
			DebugMsg := 'Empty ITC message received.';
			fbDebugMsg.M_SendErrorMsg(DebugMsg);
			
		(*******************************************************************************
		  Add TU data
		********************************************************************************)
		E_ITC_MsgTypeConv.E_ADD_TU_REQUEST:
			M_ITC_ATQ(meChannelSrc := meChannelSrc, mpData := mpData, mLen := mLen);
			
		(*******************************************************************************
		  Remove TU data
		********************************************************************************)
		E_ITC_MsgTypeConv.E_REMOVE_TU_REQUEST:
			M_ITC_RTQ(meChannelSrc := meChannelSrc, mpData := mpData, mLen := mLen);
			
		(*******************************************************************************
		  Modify error 
		********************************************************************************)
		E_ITC_MsgTypeConv.E_ERROR_REQUEST:
			M_ITC_ERQ(meChannelSrc := meChannelSrc, mpData := mpData, mLen := mLen);

	ELSE
		// Unknown ITC message type received
		DebugMsg := CONCAT('Function emulation unknown ITC Message type: ', INT_TO_STRING(FunctionBase.eMsgType));
		fbDebugMsg.M_SendErrorMsg(DebugMsg);
	END_CASE
END_IF
END_METHOD

METHOD PRIVATE M_ITC_RTQ : BOOL
VAR_INPUT
	meChannelSrc		: E_MFCS_CHANNEL; // Number of the source 
	mpData				: PVOID; // Data  pointer 
	mLen				: UDINT; // Data length
END_VAR
// Map data
F_BlockCopy(
	pSrc:= mpData, 
	LenSrc:= mLen, 
	pDest:= ADR(FunctionBase.Data), 
	LenDest:= SIZEOF(FunctionBase.Data));

// If a valid zone number is ready
IF FunctionBase.Data.ZoneNumber > 0 THEN
	// Send "Remove TU" request to zone
	ZoneData[FunctionBase.Data.ZoneNumber].ITC.Commands.RemoveTU := TRUE;
	ZoneData[FunctionBase.Data.ZoneNumber].ITC.Commands.IndexToRemove := FunctionBase.IndexToRemove[FunctionBase.Data.ZoneNumber];
ELSE
	// Invalid zone number
	DebugMsg := 'REMOVE_TU_DATA - No valid ZoneNumber, request rejected';
	fbDebugMsg.M_SendErrorMsg(DebugMsg);
END_IF
END_METHOD

METHOD M_MoveTU_DataIndex : DINT;
VAR_INPUT
	mZoneNumber : INT;
END_VAR
// Return current TU-data index
M_MoveTU_dataIndex := ZoneData[mZoneNumber].TransportControlData.TU_DataIndex;
// Update last TU-data index
ZoneData[mZoneNumber].TransportControlData.LastTU_DataIndex := M_MoveTU_dataIndex;
// Delete current TU-data index
ZoneData[mZoneNumber].TransportControlData.TU_DataIndex := 0;
// Reset data present
ZoneData[mZoneNumber].TransportControlData.DataPresent := FALSE;
END_METHOD

METHOD M_SetHW_Inputs : BOOL
(**************************************************************************************
 * 	Application		:	BoxControl Framework
 *	Revision		:	$Revision: 461869 $
 *	Revision date	:	$Date: 2020-09-25 14:40:24 +0200 (fre, 25 sep 2020) $
 *	Last changed by	:	$Author: d7mangc $
 *	URL				:	$URL: http://almscdc.swisslog.com/repo/SWPD/Development/BoxControlFramework/20_Release/tags/R1.12.0/01_Software/BCF/BCF/JumpStart/20_Product/10_BCF/11_Conv/12_E_Functions/09_Emulation/FB_FunctionConvEmulation.TcPOU $
 *
 *	Purpose			:	Base set HW inputs, needs to be overriden from inheritance object
 *
 * ------------------------------------------------------------------------------------
 *	Copyright Swisslog [IP AG], Switzerland. All rights reserved.
 * 
 * ------------------------------------------------------------------------------------
 *	
 * 	Revision History: 
 *
 * 	VERSION			DATE			INITIALS			DESCRIPTION
 *	0.1				01.01.2001		swl					Example
 *
 **************************************************************************************)
VAR_INPUT
	mZoneNumber : INT; // Zone number
	mSetHW_Input : ST_SetHW_Inputs; // Set HW inputs state
	mEnableHW_Input : ST_SetHW_Inputs; // Enable HW inputs for processing
END_VAR
;
END_METHOD

METHOD M_UpdateRealObjectData
(**************************************************************************************
 * 	Application		:	BoxControl Framework
 *	Revision		:	$Revision: 461869 $
 *	Revision date	:	$Date: 2020-09-25 14:40:24 +0200 (fre, 25 sep 2020) $
 *	Last changed by	:	$Author: d7mangc $
 *	URL				:	$URL: http://almscdc.swisslog.com/repo/SWPD/Development/BoxControlFramework/20_Release/tags/R1.12.0/01_Software/BCF/BCF/JumpStart/20_Product/10_BCF/11_Conv/12_E_Functions/09_Emulation/FB_FunctionConvEmulation.TcPOU $
 *
 *	Purpose			:	This methode gets always the current values of the real object
 *
 * ------------------------------------------------------------------------------------
 *	Copyright Swisslog [IP AG], Switzerland. All rights reserved.
 * 
 * ------------------------------------------------------------------------------------
 *	
 * 	Revision History: 
 *
 * 	VERSION			DATE			INITIALS			DESCRIPTION
 *	0.1				01.01.2001		swl					Example
 *
 **************************************************************************************)

IF __ISVALIDREF(FunctionRegistry[eFunctionNumber].rFunctionData) THEN
	FunctionBase.rFunctionDataReal	REF= FunctionRegistry[eFunctionNumber].rFunctionData;
ELSE
	FunctionBase.rFunctionDataReal REF= FunctionBase.FunctionDataEmpty;
END_IF

IF __ISVALIDREF(FunctionRegistry[eFunctionNumber].rFunctionInterface) THEN
	FunctionBase.rFunctionInterfaceReal REF= FunctionRegistry[eFunctionNumber].rFunctionInterface;
ELSE
	FunctionBase.rFunctionInterfaceReal REF= FunctionBase.FunctionInterfaceEmpty;
END_IF

IF __ISVALIDREF(FunctionRegistry[eFunctionNumber].rFunction) THEN
	FunctionBase.rZoneDataReal	REF= FunctionRegistry[eFunctionNumber].rFunction.ZoneData;
ELSE
	FunctionBase.rZoneDataReal REF= FunctionBase.ZoneDataEmpty;
END_IF

IF __ISVALIDREF(FunctionRegistry[eFunctionNumber].rFunction) THEN
	FunctionBase.rZoneInterfaceReal REF= FunctionRegistry[eFunctionNumber].rFunction.ZoneInterface;
ELSE
	FunctionBase.rZoneInterfaceReal REF= FunctionBase.ZoneInterfaceEmpty;
END_IF

IF __ISVALIDREF(FunctionRegistry[eFunctionNumber].rSettingsFunction) THEN
	FunctionBase.rSettingsFunctionReal REF= FunctionRegistry[eFunctionNumber].rSettingsFunction;
ELSE
	FunctionBase.rSettingsFunctionReal REF= FunctionBase.SettingsEmpty;
END_IF
END_METHOD

END_FUNCTION_BLOCK

// ---- 20_Product/10_BCF/11_Conv/12_E_Functions/10_Helper/F_IsFunctionInitialized.TcPOU
FUNCTION F_IsFunctionInitialized : BOOL
(**************************************************************************************
 * 	Application		:	BoxControl Framework
 *	Revision		:	$Revision: 404529 $
 *	Revision date	:	$Date: 2018-04-23 08:21:38 +0200 (Mo., 23 Apr 2018) $
 *	Last changed by	:	$Author: b7bolm $
 *	URL				:	$URL: http://almscdc.swisslog.com/repo/SWPD/Development/BoxControlFramework/20_Release/trunk/01_Software/BCF/BCF/JumpStart/20_Product/10_App/12_E_Functions/10_Lib/10_Conv/10_Functions/F_IsFunctionInitialized.TcPOU $
 *
 *	Purpose			:	Returns function base data
 *
 * ------------------------------------------------------------------------------------
 *	Copyright Swisslog [IP AG], Switzerland. All rights reserved.
 * 
 * ------------------------------------------------------------------------------------
 *	
 * 	Revision History: 
 *
 * 	VERSION			DATE			INITIALS			DESCRIPTION
 *	0.1				01.01.2001		swl					Example
 *
 **************************************************************************************)
VAR_INPUT
	eFunctionNumber			: E_FunctionNumber; // Element function Number
END_VAR

VAR
	FunctionReg				: ST_FunctionRegistryConv;
END_VAR


// Check if function number is valid
IF eFunctionNumber > E_FunctionNumber.F_BEGIN_FUNCTION AND
   eFunctionNumber < E_FunctionNumber.F_END_FUNCTION THEN

	// Check reference is valid
	IF __ISVALIDREF(FunctionRegistry[eFunctionNumber].rFunctionData) THEN
   		// Return function data
   		F_IsFunctionInitialized := FunctionRegistry[eFunctionNumber].rFunctionData.Init;
	END_IF
END_IF

END_FUNCTION

// ---- 20_Product/10_BCF/11_Conv/12_E_Functions/10_Helper/FB_DistanceMeter.TcPOU
FUNCTION_BLOCK FB_DistanceMeter
(**************************************************************************************
 * 	Application		:	BoxControl Framework
 *	Revision		:	$Revision: 475083 $
 *	Revision date	:	$Date: 2021-04-10 12:07:10 +0200 (lör, 10 apr 2021) $
 *	Last changed by	:	$Author: d7mangc $
 *	URL				:	$URL: http://almscdc.swisslog.com/repo/SWPD/Development/BoxControlFramework/20_Release/tags/R1.12.0/01_Software/BCF/BCF/JumpStart/20_Product/10_BCF/11_Conv/12_E_Functions/10_Helper/FB_DistanceMeter.TcPOU $
 *
 *	Purpose			:	Distance meter based on encoder value
 *						
 *
 * ------------------------------------------------------------------------------------
 *	Copyright Swisslog [IP AG], Switzerland. All rights reserved.
 * 
 * ------------------------------------------------------------------------------------
 *	
 * 	Revision History: 
 *
 * 	VERSION			DATE			INITIALS			DESCRIPTION
 *	0.1				01.01.2001		swl					Example
 *
 **************************************************************************************)
VAR_INPUT
	Run					: BOOL;
	EncoderValue		: WORD;
	SetPoint			: DINT;
	PresetDistance		: DINT;
	Input_TU_DataIndex	: DINT;
END_VAR

VAR_OUTPUT
	Q					: BOOL;
	Distance			: DINT;
	TU_DataIndex		: DINT;
END_VAR

VAR
	Trg			     : BOOL; // Trigger detection for start signal
	LastEncoderValue : WORD;
	Inc 			 : INT;
END_VAR

IF Run THEN
	// Detect start trigger and preset values
	IF NOT Trg AND Run THEN
		LastEncoderValue := EncoderValue;
		Distance := PresetDistance;
		TU_DataIndex := Input_TU_DataIndex;
	END_IF
	
	// Calculate increment
	IF EncoderValue >= LastEncoderValue THEN
		Inc := WORD_TO_INT(EncoderValue - LastEncoderValue);
	// Handle overflow
	ELSE
		Inc := WORD_TO_INT(EncoderValue + 1 + 16#FFFF - LastEncoderValue);
	END_IF	

	// Update last encoder value
	LastEncoderValue := EncoderValue;
	
	// Update outputs
	IF NOT Q THEN
		Distance := Distance + ABS(Inc);
		IF Distance >= SetPoint THEN
			Q := TRUE;
		END_IF
	END_IF
ELSE
	// Reset outputs
	Q := FALSE;
	TU_DataIndex := 0;
END_IF

Trg := Run;

// Changes the current position (distance)
METHOD PUBLIC M_SetDistance

VAR_INPUT
	NewDistance 	: DINT	:= 0;
END_VAR
IF Run THEN
	Distance := NewDistance;
	THIS^();
END_IF
END_METHOD

END_FUNCTION_BLOCK

// ---- 20_Product/10_BCF/11_Conv/12_E_Functions/10_Helper/FB_GetDistance.TcPOU
FUNCTION_BLOCK FB_GetDistance  
(**************************************************************************************
 * 	Application		:	BoxControl Framework
 *	Revision		:	$Revision: 404529 $
 *	Revision date	:	$Date: 2018-04-23 08:21:38 +0200 (Mo., 23 Apr 2018) $
 *	Last changed by	:	$Author: b7bolm $
 *	URL				:	$URL: http://almscdc.swisslog.com/repo/SWPD/Development/BoxControlFramework/20_Release/trunk/01_Software/BCF/BCF/JumpStart/20_Product/10_App/12_E_Functions/10_Lib/10_Conv/10_Functions/FB_GetDistance.TcPOU $
 *
 *	Purpose			:	Meauseres the distance in increments and mm between two sensors.
 * 						
 *
 * ------------------------------------------------------------------------------------
 *	Copyright Swisslog [IP AG], Switzerland. All rights reserved.
 * 
 * ------------------------------------------------------------------------------------
 *	
 * 	Revision History: 
 *
 * 	VERSION			DATE			INITIALS			DESCRIPTION
 *	0.1				01.01.2001		swl					Example
 *
 **************************************************************************************)

VAR_INPUT
	StartSignal	: BOOL; // Start measurement
	EndSignal	: BOOL; // Stop measurement
	EncoderValue: DINT; // Actual encoder position
	Resolution	: DINT; // Encoder resolution inc/m
END_VAR

VAR_OUTPUT
	Distance_Inc: DINT; // Distance in increments meausered between the two sensors.
	Distance_mm	: DINT; // Distance in mm meausered between the two sensors.
END_VAR

VAR
	StartMeasurementTrig	: R_TRIG; // Trigger
	EndMeasurementTrig		: R_TRIG; // Trigger
	StartPosition			: DINT;	// Startposition in increments
	EndPosition				: DINT; // Endposition in increments
END_VAR


// Wait for TU front edge on start signal
StartMeasurementTrig(clk := StartSignal);
IF StartMeasurementTrig.Q THEN
	StartPosition := EncoderValue;
END_IF

// Wait for TU front edge at conveyor end signal
EndMeasurementTrig(clk := EndSignal);
IF EndMeasurementTrig.Q THEN
	EndPosition := EncoderValue;
	// Handle Overflow 
	IF EndPosition >= StartPosition THEN
		// Calculate distance in increments
		Distance_Inc := EndPosition - StartPosition;
	ELSE
		Distance_Inc := 0;	
	END_IF	
	// Calculat distance in [mm]
	IF Resolution > 0 THEN
		Distance_mm := REAL_TO_DINT(DINT_TO_REAL(Distance_Inc) / DINT_TO_REAL(Resolution) * 1000.0);
	END_IF
END_IF

END_FUNCTION_BLOCK

// ---- 20_Product/10_BCF/11_Conv/12_E_Functions/10_Helper/FB_GetEncoderResolution.TcPOU
/// Uses two defined signals to determine encoder resolution
/// Remark: A constant speed is requirement for the movement between the signals, to get an accurat result
/// Remark: Drive direction has to be according order of Signal 1 and Signal 2
FUNCTION_BLOCK FB_GetEncoderResolution  
(************************************************************************************** 
* 	Application 		: BoxControl Framework 
* 	Revision 			: $Revision: 408723 $ 
* 	Revision date 		: $Date: 2018-06-27 13:49:08 +0200 (Wed, 27 Jun 2018) $ 
* 	Last changed by 	: $Author: b7bolm $ 
* 	URL 				: $URL: http://almscdc.swisslog.com/repo/SWPD/Development/BoxControlFramework/21_Projects/BCF_2.0/trunk/BCF/BCF/JumpStart/20_Product/10_App/12_E_Functions/10_Lib/10_Conv/FB_FunctionList.TcPOU $ 
* ------------------------------------------------------------------------------------ 
* 	© Swisslog AG 
* 	Swisslog is not liable for any usage of this source code that is not agreed 
* 	on between Swisslog and the other party. The mandatory legal liability remains 
* 	unaffected. 
* ------------------------------------------------------------------------------------ 
* 	Revision History: 
*
*  VERSION DATE         INITIALS     DESCRIPTION
*  0.0     DD.MM.YYYY   (name)       (explain customized modifications)
* 
**************************************************************************************)
VAR_INPUT
	Run						: BOOL; // Rising edge starts measurement and resets outputs
	StartSignal				: BOOL; // Start measurement
	EndSignal				: BOOL; // Stop measurement
	DistanceSignals			: UINT; // Distance between start and end signal [mm]
	EncoderValue			: ULINT; // Encoder values [increment]
	EncoderFW_Desc			: BOOL := FALSE; // Encoder counts in descending sequence 9,8,7,6... to move forward
	MaxEncoderValue			: UDINT; // Max value of input "EncoderValue" Remark: Used to detect overflow, needs to be less than DINT size [increment]
END_VAR

VAR_OUTPUT
	Busy					: BOOL; // Measurement running
	DistanceInc				: ULINT; // Distance in increments meausered between the two sensors.
	Resolution				: REAL; // Encoder resolution in increment per milimeter [inc/mm]
	Error					: BOOL; // Overflow during measurement or input value error
END_VAR

VAR
	DeltaEncoderValue		: LINT; // Delta encoder value (LastValue - CurrentValue)
	TrackingEncoderValue	: ULINT; // Internal encoder of traveled increments [increment]
	RunTrig					: R_TRIG; // Run trigger to start measurement and reset
	StartMeasurementTrig	: R_TRIG; // Start signal for measurement
	EndMeasurementTrig		: R_TRIG; // End of measurement
	LastEncoderValue		: ULINT; // Last encoder value [increment]
	LastTrackingEncoderValue: ULINT; // Last tracking encoder value [increment]
	StartPosition			: ULINT; // Startposition in increments [increment]
	EndPosition				: ULINT; // Endposition in increments [increment]
END_VAR

// Start measurment and initialize values
RunTrig(clk := Run);
IF RunTrig.Q THEN
	DistanceInc := 0;
	Resolution := 0;
	StartPosition := 0;
	EndPosition := 0;
	DeltaEncoderValue := 0;
	TrackingEncoderValue := 0;
	
	// Check inputs
	IF DistanceSignals = 0 THEN
		Error := TRUE;
	ELSE
		Busy := TRUE;
		Error := FALSE;
	END_IF
END_IF

// When measurement is running, wait for start and end signal
IF Busy AND Run THEN
	// Create internal encoder to make movement independent from encoder overflow
	DeltaEncoderValue := ULINT_TO_LINT(EncoderValue) - ULINT_TO_LINT(LastEncoderValue);
	
	IF ABS(DeltaEncoderValue) > MaxEncoderValue/2 THEN
		// Correction with + 1 is to include the 0 in MaxEncoderValue
		IF DeltaEncoderValue < 0 THEN
			DeltaEncoderValue := DeltaEncoderValue + UDINT_TO_LINT(MaxEncoderValue) + 1;
		ELSE
			DeltaEncoderValue := - ULINT_TO_LINT(EncoderValue) - ULINT_TO_LINT(LastEncoderValue) + UDINT_TO_LINT(MaxEncoderValue) - 1;
		END_IF
	END_IF
	
	LastEncoderValue := EncoderValue;
	
	IF EncoderFW_Desc THEN
		TrackingEncoderValue := TrackingEncoderValue - LINT_TO_ULINT(DeltaEncoderValue);
	ELSE
		TrackingEncoderValue := TrackingEncoderValue + LINT_TO_ULINT(DeltaEncoderValue);
	END_IF
	
	LastEncoderValue := EncoderValue;
	LastTrackingEncoderValue := TrackingEncoderValue;

	// Internal overflow, error
	IF TrackingEncoderValue < LastTrackingEncoderValue THEN
		Error := TRUE;
		Busy := FALSE;
		RETURN;
	END_IF

	// Wait for front edge
	StartMeasurementTrig(clk := StartSignal);
	
	IF StartMeasurementTrig.Q THEN
		StartPosition := TrackingEncoderValue;
	END_IF
	
	// Wait for rear edge
	EndMeasurementTrig(clk := EndSignal);
	
	IF EndMeasurementTrig.Q THEN
		EndPosition := TrackingEncoderValue;
		
		IF EndPosition >= StartPosition THEN
			DistanceInc := EndPosition - StartPosition;
			Resolution := ULINT_TO_REAL(DistanceInc) / UINT_TO_REAL(DistanceSignals);
		// Otherwise overflow, distance greather than data type LINT 
		ELSE
			Error := TRUE;
		END_IF
		
		Busy := FALSE;
	END_IF
ELSIF Busy THEN
	Busy := FALSE;
	Error := TRUE;
END_IF

END_FUNCTION_BLOCK

// ---- 20_Product/10_BCF/11_Conv/12_E_Functions/10_Helper/FB_Handover.TcPOU
/// Basic handover implementation
FUNCTION_BLOCK FB_Handover
(************************************************************************************** 
* 	Application 		: BoxControl Framework 
* 	Revision 			: $Revision: 408723 $ 
* 	Revision date 		: $Date: 2018-06-27 13:49:08 +0200 (Wed, 27 Jun 2018) $ 
* 	Last changed by 	: $Author: b7bolm $ 
* 	URL 				: $URL: http://almscdc.swisslog.com/repo/SWPD/Development/BoxControlFramework/21_Projects/BCF_2.0/trunk/BCF/BCF/JumpStart/20_Product/10_App/12_E_Functions/10_Lib/10_Conv/FB_FunctionList.TcPOU $ 
* ------------------------------------------------------------------------------------ 
* 	© Swisslog AG 
* 	Swisslog is not liable for any usage of this source code that is not agreed 
* 	on between Swisslog and the other party. The mandatory legal liability remains 
* 	unaffected. 
* ------------------------------------------------------------------------------------ 
* 	Revision History: 
* 
* 	VERSION 		DATE 			INITIALS 			DESCRIPTION 
* 	0.1 			22.08.2018 		herzig 				First implementation
*	0.2				05.10.2018		b7bolm				Review
* 
**************************************************************************************)
VAR_INPUT
	Enable						: BOOL; // Allow handover in general  
	RequestHandover				: BOOL; // Rising edge initiates a new transport
	NextZonePresent 			: BOOL;	// Next zone is known
	HandoverComplete			: BOOL; // Handover complete
	DriveReady					: BOOL; // Drive is ready to be switched on
	iListener 					: I_HandoverListener; // Listener for any handover events
END_VAR
VAR_OUTPUT
	FastSpeed					: BOOL; // Fastspeed possible
	DriveRun					: BOOL; // Switch drive on
	DriveRequest				: BOOL; // Request drive 
	eHandOverState				: E_HandOverState; // Handover state
	eNextTakeOverState			: E_TakeOverState; // Next takeover state
	RequestNextTransportData 	: BOOL; // Request next transport data
	DeleteNextTransportData 	: BOOL; // Delete next transport data
	HandoverOngoing				: BOOL; // Handover ongoing, interface in interaction
END_VAR
VAR_IN_OUT
	NextTransportData			: ST_TransportData; // Next transport data
	ErrorData					: ST_ErrorDataSet;
END_VAR
VAR
	CompleteReceived			: BOOL; // Complete received
END_VAR

// To ensure not missing any complete message during state change
IF HandoverComplete THEN
	CompleteReceived := HandoverComplete;
END_IF

// Handover state machine
CASE eHandOverState OF
	// Idle
	E_HandOverState.IDLE:
		DeleteNextTransportData := FALSE;
		RequestNextTransportData := FALSE;
		DriveRequest := FALSE;
		DriveRun := FALSE;
		CompleteReceived := FALSE;

		IF RequestHandover THEN
			// Transport is released, no command to stop or error active
			IF Enable AND
			   NOT HandoverComplete AND
			   ErrorData.ErrorType <> E_ErrorType.ERROR THEN
				 
				// If next zone or function is available
				IF NextZonePresent THEN	
					DriveRequest := NOT DriveReady;
					eHandOverState := E_HandOverState.READY;
				ELSE
					RequestNextTransportData := TRUE;
				END_IF
			END_IF
		END_IF

  	// Ready
	E_HandOverState.READY:	
		DriveRequest := NOT DriveReady;
	
		IF NOT Enable OR NOT RequestHandover OR
		   ErrorData.ErrorType = E_ErrorType.ERROR OR
           NOT NextZonePresent OR HandoverComplete THEN
			
			DeleteNextTransportData := TRUE;   
			eHandOverState := E_HandOverState.IDLE;
			
		// Next position started takeover
		ELSIF NextTransportData.rTransportControlData.eTakeOverState = E_TakeOverState.ACTIVE THEN			
			IF iListener <> 0 THEN
			   iListener.M_HandoverStartEvent();
		   	END_IF
		
			// Set start drive
			DriveRun := TRUE;
			eHandOverState := E_HandOverState.ACTIVE;
		END_IF
		
 	// Active
	E_HandOverState.ACTIVE:
		DriveRequest := NOT DriveReady;
		DriveRun := TRUE;

		// Stop handover
		IF NOT Enable OR
		   ErrorData.ErrorType = E_ErrorType.ERROR OR 
           NOT DriveReady THEN   
			DriveRun := FALSE;
			eHandOverState := E_HandOverState.STOP;
	
		ELSIF CompleteReceived THEN
			DriveRun := FALSE;
			
			IF iListener <> 0 THEN
				iListener.M_HandoverCompleteEvent();
			END_IF
			
			eHandOverState := E_HandOverState.COMPLETE;	
			
		// If next position stopped handover
		ELSIF NextTransportData.rTransportControlData.eTakeOverState = E_TakeOverState.STOP THEN
			DriveRun := FALSE;
			eHandOverState := E_HandOverState.INTERRUPTED;

		// If the next position aborted the handover or the link is broken
		ELSIF NextTransportData.rTransportControlData.eTakeOverState = E_TakeOverState.IDLE OR
			  NextTransportData.rTransportControlData.eTakeOverState = E_TakeOverState.UNDEFINED THEN  
			DeleteNextTransportData := TRUE;
			DriveRun := FALSE;
			eHandOverState := E_HandOverState.IDLE;
			
		// Next position completed takeover (normal completion with MFC)
		ELSIF NextTransportData.rTransportControlData.eTakeOverState = E_TakeOverState.COMPLETE THEN
			DeleteNextTransportData := TRUE;
			
			DriveRun := FALSE;
			eHandOverState := E_HandOverState.IDLE;
		END_IF

  	// Stop
	E_HandOverState.STOP:
		// If the next position aborted the takeover or the link is broken, cancel the started handover
		IF NextTransportData.rTransportControlData.eTakeOverState = E_TakeOverState.IDLE OR
		   NextTransportData.rTransportControlData.eTakeOverState = E_TakeOverState.UNDEFINED THEN
		   	DriveRun := FALSE;
			DeleteNextTransportData := TRUE;
			eHandOverState := E_HandOverState.IDLE;

		// If transport is enabled and position is started
		ELSIF Enable THEN
			// If no error is pending
			IF ErrorData.ErrorType <> E_ErrorType.ERROR THEN
				IF DriveReady THEN
					DriveRun := TRUE;
					DriveRequest := FALSE;
					eHandOverState := E_HandOverState.ACTIVE;
				ELSE
					DriveRequest := TRUE;
				END_IF
			END_IF
		END_IF

  	// Interrupted
	E_HandOverState.INTERRUPTED:
		// If the next position aborted the takeover or the link is broken, cancel the started handover
		IF NextTransportData.rTransportControlData.eTakeOverState = E_TakeOverState.IDLE OR
		   NextTransportData.rTransportControlData.eTakeOverState = E_TakeOverState.UNDEFINED THEN
			DeleteNextTransportData := TRUE;
			eHandOverState := E_HandOverState.IDLE;

		// If the next position is active again
		ELSIF NextTransportData.rTransportControlData.eTakeOverState = E_TakeOverState.ACTIVE THEN
			DriveRun := TRUE;
			eHandOverState := E_HandOverState.ACTIVE;
		END_IF
		
  	// Complete
	E_HandOverState.COMPLETE:	
		// No pending transfer -> change to idle
		IF NextTransportData.rTransportControlData.eTakeOverState = E_TakeOverState.COMPLETE OR
		   NextTransportData.rTransportControlData.eTakeOverState = E_TakeOverState.READY OR
		   NextTransportData.rTransportControlData.eTakeOverState = E_TakeOverState.IDLE OR
		   NextTransportData.rTransportControlData.eTakeOverState = E_TakeOverState.UNDEFINED THEN
			DeleteNextTransportData := TRUE;

			eHandOverState := E_HandOverState.IDLE;
		END_IF
ELSE
	// Set error
	F_SetError(	
		ErrorType	:= E_ErrorType.ERROR,
		ErrorParam	:= INT_TO_STRING(eHandOverState),
		ErrorMsg	:= E_ErrorConv.SOFTWARE_ERROR,
		ErrorData	:= ErrorData);
END_CASE

// When a handover is ongoing
IF DriveRun THEN
	// During handover follow next position
	FastSpeed := NextTransportData.rTransportControlData.FastSpeedActive;
	
// Otherwise, fast speed is dependet if next position is available for takeover
ELSE
	FastSpeed := (RequestHandover AND NextTransportData.rTransportControlData.eTakeoverState = E_TakeOverState.READY) OR
				  NOT RequestHandover;
END_IF

eNextTakeOverState := NextTransportData.rTransportControlData.eTakeOverState;

HandoverOngoing := eHandOverState = E_HandoverState.ACTIVE OR
				   eHandOverState = E_HandoverState.STOP OR
				   eHandOverState = E_HandoverState.INTERRUPTED;

